LIN {X 0,Y 509.293,Z 778.89,A -85,B 0,C 180,E1 -5495.543,E2 -5495.543} C_VEL
LIN {X 0,Y 509.338,Z 774.921,A -85,B 0,C 180,E1 -5496.696,E2 -5496.696} C_VEL
LIN {X 0,Y 509.453,Z 769.669,A -85,B 0,C 180,E1 -5497.929,E2 -5497.929} C_VEL
LIN {X 0,Y 509.604,Z 763.492,A -85,B 0,C 180,E1 -5499.125,E2 -5499.125} C_VEL
LIN {X 0,Y 509.79,Z 757.418,A -85,B 0,C 180,E1 -5500.123,E2 -5500.123} C_VEL
LIN {X 0,Y 510.074,Z 750.342,A -85,B 0,C 180,E1 -5501.122,E2 -5501.122} C_VEL
LIN {X 0,Y 510.293,Z 742.434,A -85,B 0,C 180,E1 -5502.082,E2 -5502.082} C_VEL
LIN {X 0,Y 510.609,Z 734.391,A -85,B 0,C 180,E1 -5502.924,E2 -5502.924} C_VEL
LIN {X 0,Y 510.98,Z 725.51,A -85,B 0,C 180,E1 -5503.724,E2 -5503.724} C_VEL
LIN {X 0,Y 511.277,Z 716.451,A -85,B 0,C 180,E1 -5504.427,E2 -5504.427} C_VEL
LIN {X 0,Y 511.699,Z 705.64,A -85,B 0,C 180,E1 -5505.127,E2 -5505.127} C_VEL
LIN {X 0,Y 512.044,Z 695.376,A -85,B 0,C 180,E1 -5505.677,E2 -5505.677} C_VEL
LIN {X 0,Y 512.33,Z 684.979,A -85,B 0,C 180,E1 -5506.131,E2 -5506.131} C_VEL
LIN {X 0,Y 512.62,Z 672.99,A -85,B 0,C 180,E1 -5506.533,E2 -5506.533} C_VEL
LIN {X 0,Y 512.826,Z 661.767,A -85,B 0,C 180,E1 -5506.802,E2 -5506.802} C_VEL
LIN {X 0,Y 513.111,Z 631.655,A -85,B 0,C 180,E1 -5507.254,E2 -5507.254} C_VEL
LIN {X 0,Y 513.563,Z 539.81,A -85,B 0,C 180,E1 -5508.56,E2 -5508.56} C_VEL
LIN {X 0,Y 510.7,Z 525.355,A -85,B 0,C 180,E1 -5508.892,E2 -5508.892} C_VEL
LIN {X 0,Y 510.69,Z 524.406,A -85,B 0,C 180,E1 -5509.004,E2 -5509.004} C_VEL
LIN {X 0,Y 511.189,Z 507.71,A -85,B 0,C 180,E1 -5512.002,E2 -5512.002} C_VEL
LIN {X 0,Y 511.684,Z 492.965,A -85,B 0,C 180,E1 -5514.662,E2 -5514.662} C_VEL
LIN {X 0,Y 511.823,Z 486.597,A -85,B 0,C 180,E1 -5515.846,E2 -5515.846} C_VEL
LIN {X 0,Y 509.91,Z 476.204,A -85,B 0,C 180,E1 -5517.944,E2 -5517.944} C_VEL
LIN {X 0,Y 509.845,Z 476.085,A -85,B 0,C 180,E1 -5520.665,E2 -5520.665} C_VEL
LIN {X 0,Y 509.859,Z 476.102,A -85,B 0,C 180,E1 -5523.46,E2 -5523.46} C_VEL
LIN {X 0,Y 509.822,Z 476.077,A -85,B 0,C 180,E1 -5526.352,E2 -5526.352} C_VEL
LIN {X 0,Y 509.845,Z 476.1,A -85,B 0,C 180,E1 -5529.351,E2 -5529.351} C_VEL
LIN {X 0,Y 509.845,Z 476.094,A -85,B 0,C 180,E1 -5532.487,E2 -5532.487} C_VEL
LIN {X 0,Y 509.853,Z 476.102,A -85,B 0,C 180,E1 -5535.331,E2 -5535.331} C_VEL
LIN {X 0,Y 509.859,Z 476.093,A -85,B 0,C 180,E1 -5538.575,E2 -5538.575} C_VEL
LIN {X 0,Y 509.846,Z 476.096,A -85,B 0,C 180,E1 -5541.786,E2 -5541.786} C_VEL
LIN {X 0,Y 509.841,Z 476.098,A -85,B 0,C 180,E1 -5544.622,E2 -5544.622} C_VEL
LIN {X 0,Y 509.859,Z 476.098,A -85,B 0,C 180,E1 -5547.48,E2 -5547.48} C_VEL
LIN {X 0,Y 509.852,Z 476.096,A -85,B 0,C 180,E1 -5550.273,E2 -5550.273} C_VEL
LIN {X 0,Y 509.88,Z 476.09,A -85,B 0,C 180,E1 -5552.944,E2 -5552.944} C_VEL
LIN {X 0,Y 509.863,Z 476.1,A -85,B 0,C 180,E1 -5555.573,E2 -5555.573} C_VEL
LIN {X 0,Y 509.814,Z 476.096,A -85,B 0,C 180,E1 -5558.148,E2 -5558.148} C_VEL
LIN {X 0,Y 509.857,Z 476.091,A -85,B 0,C 180,E1 -5560.681,E2 -5560.681} C_VEL
LIN {X 0,Y 509.879,Z 476.098,A -85,B 0,C 180,E1 -5563.174,E2 -5563.174} C_VEL
LIN {X 0,Y 509.854,Z 476.092,A -85,B 0,C 180,E1 -5565.634,E2 -5565.634} C_VEL
LIN {X 0,Y 509.904,Z 476.089,A -85,B 0,C 180,E1 -5568.874,E2 -5568.874} C_VEL
LIN {X 0,Y 509.943,Z 476.083,A -85,B 0,C 180,E1 -5572.078,E2 -5572.078} C_VEL
LIN {X 0,Y 509.974,Z 476.07,A -85,B 0,C 180,E1 -5574.464,E2 -5574.464} C_VEL
LIN {X 0,Y 510.046,Z 476.078,A -85,B 0,C 180,E1 -5577.631,E2 -5577.631} C_VEL
LIN {X 0,Y 510.056,Z 476.066,A -85,B 0,C 180,E1 -5580.789,E2 -5580.789} C_VEL
LIN {X 0,Y 509.95,Z 476.078,A -85,B 0,C 180,E1 -5583.16,E2 -5583.16} C_VEL
LIN {X 0,Y 509.968,Z 476.081,A -85,B 0,C 180,E1 -5586.329,E2 -5586.329} C_VEL
LIN {X 0,Y 509.909,Z 476.084,A -85,B 0,C 180,E1 -5588.72,E2 -5588.72} C_VEL
LIN {X 0,Y 509.895,Z 476.093,A -85,B 0,C 180,E1 -5591.931,E2 -5591.931} C_VEL
LIN {X 0,Y 509.883,Z 476.096,A -85,B 0,C 180,E1 -5595.242,E2 -5595.242} C_VEL
LIN {X 0,Y 509.878,Z 476.092,A -85,B 0,C 180,E1 -5598.001,E2 -5598.001} C_VEL
LIN {X 0,Y 509.841,Z 476.098,A -85,B 0,C 180,E1 -5601.002,E2 -5601.002} C_VEL
LIN {X 0,Y 509.86,Z 476.088,A -85,B 0,C 180,E1 -5604.426,E2 -5604.426} C_VEL
LIN {X 0,Y 509.878,Z 476.094,A -85,B 0,C 180,E1 -5607.056,E2 -5607.056} C_VEL
LIN {X 0,Y 509.871,Z 476.094,A -85,B 0,C 180,E1 -5609.75,E2 -5609.75} C_VEL
LIN {X 0,Y 509.868,Z 476.094,A -85,B 0,C 180,E1 -5612.775,E2 -5612.775} C_VEL
LIN {X 0,Y 509.834,Z 476.102,A -85,B 0,C 180,E1 -5615.582,E2 -5615.582} C_VEL
LIN {X 0,Y 509.842,Z 476.099,A -85,B 0,C 180,E1 -5618.338,E2 -5618.338} C_VEL
LIN {X 0,Y 509.85,Z 476.096,A -85,B 0,C 180,E1 -5621.425,E2 -5621.425} C_VEL
LIN {X 0,Y 509.848,Z 476.094,A -85,B 0,C 180,E1 -5624.668,E2 -5624.668} C_VEL
LIN {X 0,Y 509.879,Z 476.092,A -85,B 0,C 180,E1 -5628.1,E2 -5628.1} C_VEL
LIN {X 0,Y 509.87,Z 476.094,A -85,B 0,C 180,E1 -5630.651,E2 -5630.651} C_VEL
LIN {X 0,Y 509.824,Z 476.095,A -85,B 0,C 180,E1 -5633.749,E2 -5633.749} C_VEL
LIN {X 0,Y 509.159,Z 476.183,A -85,B 0,C 180,E1 -5634.409,E2 -5634.409} C_VEL
LIN {X 0,Y 506.34,Z 476.537,A -85,B 0,C 180,E1 -5635.481,E2 -5635.481} C_VEL
LIN {X 0,Y 503.947,Z 476.835,A -85,B 0,C 180,E1 -5636.344,E2 -5636.344} C_VEL
LIN {X 0,Y 502.899,Z 476.964,A -85,B 0,C 180,E1 -5637.011,E2 -5637.011} C_VEL
LIN {X 0,Y 502.802,Z 476.976,A -85,B 0,C 180,E1 -5637.236,E2 -5637.236} C_VEL
LIN {X 0,Y 502.825,Z 476.978,A -85,B 0,C 180,E1 -5640.062,E2 -5640.062} C_VEL
LIN {X 0,Y 502.829,Z 476.973,A -85,B 0,C 180,E1 -5642.534,E2 -5642.534} C_VEL
LIN {X 0,Y 502.823,Z 476.975,A -85,B 0,C 180,E1 -5645.299,E2 -5645.299} C_VEL
LIN {X 0,Y 502.78,Z 476.985,A -85,B 0,C 180,E1 -5647.827,E2 -5647.827} C_VEL
LIN {X 0,Y 502.821,Z 476.976,A -85,B 0,C 180,E1 -5650.401,E2 -5650.401} C_VEL
LIN {X 0,Y 502.83,Z 476.973,A -85,B 0,C 180,E1 -5652.932,E2 -5652.932} C_VEL
LIN {X 0,Y 502.841,Z 476.974,A -85,B 0,C 180,E1 -5655.429,E2 -5655.429} C_VEL
LIN {X 0,Y 502.873,Z 476.968,A -85,B 0,C 180,E1 -5658.717,E2 -5658.717} C_VEL
LIN {X 0,Y 502.898,Z 476.97,A -85,B 0,C 180,E1 -5661.967,E2 -5661.967} C_VEL
LIN {X 0,Y 502.933,Z 476.963,A -85,B 0,C 180,E1 -5664.387,E2 -5664.387} C_VEL
LIN {X 0,Y 503.022,Z 476.953,A -85,B 0,C 180,E1 -5667.598,E2 -5667.598} C_VEL
LIN {X 0,Y 503.024,Z 476.955,A -85,B 0,C 180,E1 -5670,E2 -5670} C_VEL
LIN {X 0,Y 503.022,Z 476.953,A -85,B 0,C 180,E1 -5672.402,E2 -5672.402} C_VEL
LIN {X 0,Y 502.934,Z 476.963,A -85,B 0,C 180,E1 -5675.613,E2 -5675.613} C_VEL
LIN {X 0,Y 502.898,Z 476.97,A -85,B 0,C 180,E1 -5678.033,E2 -5678.033} C_VEL
LIN {X 0,Y 502.873,Z 476.968,A -85,B 0,C 180,E1 -5681.283,E2 -5681.283} C_VEL
LIN {X 0,Y 502.841,Z 476.974,A -85,B 0,C 180,E1 -5684.571,E2 -5684.571} C_VEL
LIN {X 0,Y 502.858,Z 476.975,A -85,B 0,C 180,E1 -5687.907,E2 -5687.907} C_VEL
LIN {X 0,Y 502.824,Z 476.976,A -85,B 0,C 180,E1 -5690.536,E2 -5690.536} C_VEL
LIN {X 0,Y 502.792,Z 476.977,A -85,B 0,C 180,E1 -5693.04,E2 -5693.04} C_VEL
LIN {X 0,Y 502.835,Z 476.975,A -85,B 0,C 180,E1 -5695.675,E2 -5695.675} C_VEL
LIN {X 0,Y 502.837,Z 476.977,A -85,B 0,C 180,E1 -5698.372,E2 -5698.372} C_VEL
LIN {X 0,Y 502.791,Z 476.978,A -85,B 0,C 180,E1 -5701.499,E2 -5701.499} C_VEL
LIN {X 0,Y 502.799,Z 476.979,A -85,B 0,C 180,E1 -5704.444,E2 -5704.444} C_VEL
LIN {X 0,Y 502.774,Z 476.969,A -85,B 0,C 180,E1 -5707.178,E2 -5707.178} C_VEL
LIN {X 0,Y 502.819,Z 476.979,A -85,B 0,C 180,E1 -5710.011,E2 -5710.011} C_VEL
LIN {X 0,Y 502.822,Z 476.963,A -85,B 0,C 180,E1 -5712.202,E2 -5712.202} C_VEL
LIN {X 0,Y 502.792,Z 476.973,A -85,B 0,C 180,E1 -5715.468,E2 -5715.468} C_VEL
LIN {X 0,Y 502.821,Z 476.976,A -85,B 0,C 180,E1 -5717.864,E2 -5717.864} C_VEL
LIN {X 0,Y 502.794,Z 476.976,A -85,B 0,C 180,E1 -5721.024,E2 -5721.024} C_VEL
LIN {X 0,Y 502.777,Z 476.979,A -85,B 0,C 180,E1 -5724.167,E2 -5724.167} C_VEL
LIN {X 0,Y 502.824,Z 476.972,A -85,B 0,C 180,E1 -5726.993,E2 -5726.993} C_VEL
LIN {X 0,Y 502.821,Z 476.97,A -85,B 0,C 180,E1 -5730.062,E2 -5730.062} C_VEL
LIN {X 0,Y 502.826,Z 476.977,A -85,B 0,C 180,E1 -5732.533,E2 -5732.533} C_VEL
LIN {X 0,Y 502.819,Z 476.965,A -85,B 0,C 180,E1 -5735.298,E2 -5735.298} C_VEL
LIN {X 0,Y 502.771,Z 476.978,A -85,B 0,C 180,E1 -5737.827,E2 -5737.827} C_VEL
LIN {X 0,Y 502.816,Z 476.977,A -85,B 0,C 180,E1 -5740.4,E2 -5740.4} C_VEL
LIN {X 0,Y 502.826,Z 476.967,A -85,B 0,C 180,E1 -5742.932,E2 -5742.932} C_VEL
LIN {X 0,Y 502.835,Z 476.969,A -85,B 0,C 180,E1 -5745.429,E2 -5745.429} C_VEL
LIN {X 0,Y 502.871,Z 476.962,A -85,B 0,C 180,E1 -5748.717,E2 -5748.717} C_VEL
LIN {X 0,Y 502.892,Z 476.96,A -85,B 0,C 180,E1 -5751.967,E2 -5751.967} C_VEL
LIN {X 0,Y 502.949,Z 476.963,A -85,B 0,C 180,E1 -5754.387,E2 -5754.387} C_VEL
LIN {X 0,Y 503.016,Z 476.937,A -85,B 0,C 180,E1 -5757.598,E2 -5757.598} C_VEL
LIN {X 0,Y 503.017,Z 476.945,A -85,B 0,C 180,E1 -5760,E2 -5760} C_VEL
LIN {X 0,Y 503.016,Z 476.954,A -85,B 0,C 180,E1 -5762.403,E2 -5762.403} C_VEL
LIN {X 0,Y 502.93,Z 476.947,A -85,B 0,C 180,E1 -5765.614,E2 -5765.614} C_VEL
LIN {X 0,Y 502.893,Z 476.962,A -85,B 0,C 180,E1 -5768.034,E2 -5768.034} C_VEL
LIN {X 0,Y 502.868,Z 476.964,A -85,B 0,C 180,E1 -5771.284,E2 -5771.284} C_VEL
LIN {X 0,Y 502.836,Z 476.969,A -85,B 0,C 180,E1 -5774.571,E2 -5774.571} C_VEL
LIN {X 0,Y 502.854,Z 476.968,A -85,B 0,C 180,E1 -5777.908,E2 -5777.908} C_VEL
LIN {X 0,Y 502.82,Z 476.971,A -85,B 0,C 180,E1 -5780.537,E2 -5780.537} C_VEL
LIN {X 0,Y 502.789,Z 476.979,A -85,B 0,C 180,E1 -5783.041,E2 -5783.041} C_VEL
LIN {X 0,Y 502.834,Z 476.968,A -85,B 0,C 180,E1 -5785.676,E2 -5785.676} C_VEL
LIN {X 0,Y 502.834,Z 476.969,A -85,B 0,C 180,E1 -5788.373,E2 -5788.373} C_VEL
LIN {X 0,Y 502.79,Z 476.974,A -85,B 0,C 180,E1 -5791.5,E2 -5791.5} C_VEL
LIN {X 0,Y 502.801,Z 476.976,A -85,B 0,C 180,E1 -5794.445,E2 -5794.445} C_VEL
LIN {X 0,Y 502.775,Z 476.976,A -85,B 0,C 180,E1 -5797.179,E2 -5797.179} C_VEL
LIN {X 0,Y 502.812,Z 476.975,A -85,B 0,C 180,E1 -5800.013,E2 -5800.013} C_VEL
LIN {X 0,Y 502.768,Z 476.982,A -85,B 0,C 180,E1 -5803.232,E2 -5803.232} C_VEL
LIN {X 0,Y 502.786,Z 476.972,A -85,B 0,C 180,E1 -5805.662,E2 -5805.662} C_VEL
LIN {X 0,Y 502.827,Z 476.968,A -85,B 0,C 180,E1 -5807.865,E2 -5807.865} C_VEL
LIN {X 0,Y 502.8,Z 476.97,A -85,B 0,C 180,E1 -5811.025,E2 -5811.025} C_VEL
LIN {X 0,Y 502.773,Z 476.957,A -85,B 0,C 180,E1 -5814.17,E2 -5814.17} C_VEL
LIN {X 0,Y 502.831,Z 476.975,A -85,B 0,C 180,E1 -5816.994,E2 -5816.994} C_VEL
LIN {X 0,Y 502.814,Z 476.967,A -85,B 0,C 180,E1 -5820.066,E2 -5820.066} C_VEL
LIN {X 0,Y 502.895,Z 477.177,A -85,B 0,C 180,E1 -5821.869,E2 -5821.869} C_VEL
LIN {X 0,Y 504.869,Z 487.556,A -85,B 0,C 180,E1 -5823.993,E2 -5823.993} C_VEL
LIN {X 0,Y 504.577,Z 499.305,A -85,B 0,C 180,E1 -5826.177,E2 -5826.177} C_VEL
LIN {X 0,Y 503.993,Z 515.407,A -85,B 0,C 180,E1 -5829.114,E2 -5829.114} C_VEL
LIN {X 0,Y 503.721,Z 524.885,A -85,B 0,C 180,E1 -5830.818,E2 -5830.818} C_VEL
LIN {X 0,Y 505.951,Z 536.372,A -85,B 0,C 180,E1 -5831.104,E2 -5831.104} C_VEL
LIN {X 0,Y 506.919,Z 541.445,A -85,B 0,C 180,E1 -5831.215,E2 -5831.215} C_VEL
LIN {X 0,Y 506.066,Z 660.21,A -85,B 0,C 180,E1 -5832.94,E2 -5832.94} C_VEL
LIN {X 0,Y 505.875,Z 671.199,A -85,B 0,C 180,E1 -5833.195,E2 -5833.195} C_VEL
LIN {X 0,Y 505.576,Z 681.524,A -85,B 0,C 180,E1 -5833.523,E2 -5833.523} C_VEL
LIN {X 0,Y 505.316,Z 691.956,A -85,B 0,C 180,E1 -5833.953,E2 -5833.953} C_VEL
LIN {X 0,Y 504.987,Z 701.932,A -85,B 0,C 180,E1 -5834.461,E2 -5834.461} C_VEL
LIN {X 0,Y 504.608,Z 711.858,A -85,B 0,C 180,E1 -5835.069,E2 -5835.069} C_VEL
LIN {X 0,Y 504.157,Z 721.586,A -85,B 0,C 180,E1 -5835.777,E2 -5835.777} C_VEL
LIN {X 0,Y 503.786,Z 731.012,A -85,B 0,C 180,E1 -5836.59,E2 -5836.59} C_VEL
LIN {X 0,Y 503.413,Z 740.042,A -85,B 0,C 180,E1 -5837.504,E2 -5837.504} C_VEL
LIN {X 0,Y 503.156,Z 747.04,A -85,B 0,C 180,E1 -5838.318,E2 -5838.318} C_VEL
LIN {X 0,Y 502.863,Z 754.543,A -85,B 0,C 180,E1 -5839.329,E2 -5839.329} C_VEL
LIN {X 0,Y 502.631,Z 761.018,A -85,B 0,C 180,E1 -5840.341,E2 -5840.341} C_VEL
LIN {X 0,Y 502.433,Z 767.557,A -85,B 0,C 180,E1 -5841.554,E2 -5841.554} C_VEL
LIN {X 0,Y 502.254,Z 772.985,A -85,B 0,C 180,E1 -5842.765,E2 -5842.765} C_VEL
LIN {X 0,Y 502.193,Z 777.426,A -85,B 0,C 180,E1 -5843.975,E2 -5843.975} C_VEL
LIN {X 0,Y 502.103,Z 780.963,A -85,B 0,C 180,E1 -5845.183,E2 -5845.183} C_VEL
LIN {X 0,Y 502.112,Z 782.9,A -85,B 0,C 180,E1 -5845.987,E2 -5845.987} C_VEL
LIN {X 0,Y 502.089,Z 785.576,A -85,B 0,C 180,E1 -5847.593,E2 -5847.593} C_VEL
LIN {X 0,Y 501.988,Z 786.858,A -85,B 0,C 180,E1 -5849.198,E2 -5849.198} C_VEL
LIN {X 0,Y 501.979,Z 787.109,A -85,B 0,C 180,E1 -5850,E2 -5850} C_VEL
LIN {X 0,Y 502.033,Z 786.388,A -85,B 0,C 180,E1 -5851.604,E2 -5851.604} C_VEL
LIN {X 0,Y 502.089,Z 785.576,A -85,B 0,C 180,E1 -5852.407,E2 -5852.407} C_VEL
LIN {X 0,Y 502.112,Z 782.9,A -85,B 0,C 180,E1 -5854.013,E2 -5854.013} C_VEL
LIN {X 0,Y 502.205,Z 778.691,A -85,B 0,C 180,E1 -5855.622,E2 -5855.622} C_VEL
LIN {X 0,Y 502.259,Z 774.722,A -85,B 0,C 180,E1 -5856.79,E2 -5856.79} C_VEL
LIN {X 0,Y 502.382,Z 769.469,A -85,B 0,C 180,E1 -5858.041,E2 -5858.041} C_VEL
LIN {X 0,Y 502.562,Z 763.293,A -85,B 0,C 180,E1 -5859.254,E2 -5859.254} C_VEL
LIN {X 0,Y 502.736,Z 757.218,A -85,B 0,C 180,E1 -5860.267,E2 -5860.267} C_VEL
LIN {X 0,Y 503.042,Z 750.142,A -85,B 0,C 180,E1 -5861.279,E2 -5861.279} C_VEL
LIN {X 0,Y 503.31,Z 742.041,A -85,B 0,C 180,E1 -5862.274,E2 -5862.274} C_VEL
LIN {X 0,Y 503.684,Z 733.132,A -85,B 0,C 180,E1 -5863.207,E2 -5863.207} C_VEL
LIN {X 0,Y 504.049,Z 724.068,A -85,B 0,C 180,E1 -5864.02,E2 -5864.02} C_VEL
LIN {X 0,Y 504.425,Z 714.786,A -85,B 0,C 180,E1 -5864.73,E2 -5864.73} C_VEL
LIN {X 0,Y 504.826,Z 705.441,A -85,B 0,C 180,E1 -5865.338,E2 -5865.338} C_VEL
LIN {X 0,Y 505.189,Z 695.177,A -85,B 0,C 180,E1 -5865.895,E2 -5865.895} C_VEL
LIN {X 0,Y 505.521,Z 684.654,A -85,B 0,C 180,E1 -5866.359,E2 -5866.359} C_VEL
LIN {X 0,Y 505.796,Z 673.229,A -85,B 0,C 180,E1 -5866.75,E2 -5866.75} C_VEL
LIN {X 0,Y 506.053,Z 661.57,A -85,B 0,C 180,E1 -5867.034,E2 -5867.034} C_VEL
LIN {X 0,Y 506.35,Z 631.458,A -85,B 0,C 180,E1 -5867.492,E2 -5867.492} C_VEL
LIN {X 0,Y 506.814,Z 540.888,A -85,B 0,C 180,E1 -5868.797,E2 -5868.797} C_VEL
LIN {X 0,Y 503.72,Z 525.076,A -85,B 0,C 180,E1 -5869.168,E2 -5869.168} C_VEL
LIN {X 0,Y 503.786,Z 522.695,A -85,B 0,C 180,E1 -5869.56,E2 -5869.56} C_VEL
LIN {X 0,Y 504.263,Z 507.55,A -85,B 0,C 180,E1 -5872.32,E2 -5872.32} C_VEL
LIN {X 0,Y 504.863,Z 491.859,A -85,B 0,C 180,E1 -5875.198,E2 -5875.198} C_VEL
LIN {X 0,Y 504.725,Z 486.455,A -85,B 0,C 180,E1 -5876.237,E2 -5876.237} C_VEL
LIN {X 0,Y 502.93,Z 477.303,A -85,B 0,C 180,E1 -5878.101,E2 -5878.101} C_VEL
LIN {X 0,Y 502.84,Z 476.965,A -85,B 0,C 180,E1 -5878.372,E2 -5878.372} C_VEL
LIN {X 0,Y 502.794,Z 476.965,A -85,B 0,C 180,E1 -5881.499,E2 -5881.499} C_VEL
LIN {X 0,Y 502.803,Z 476.976,A -85,B 0,C 180,E1 -5883.993,E2 -5883.993} C_VEL
LIN {X 0,Y 502.775,Z 476.956,A -85,B 0,C 180,E1 -5887.177,E2 -5887.177} C_VEL
LIN {X 0,Y 502.786,Z 476.977,A -85,B 0,C 180,E1 -5890.014,E2 -5890.014} C_VEL
LIN {X 0,Y 502.8,Z 476.971,A -85,B 0,C 180,E1 -5892.198,E2 -5892.198} C_VEL
LIN {X 0,Y 502.797,Z 476.981,A -85,B 0,C 180,E1 -5895.467,E2 -5895.467} C_VEL
LIN {X 0,Y 502.822,Z 476.973,A -85,B 0,C 180,E1 -5898.934,E2 -5898.934} C_VEL
LIN {X 0,Y 502.789,Z 476.973,A -85,B 0,C 180,E1 -5902.045,E2 -5902.045} C_VEL
LIN {X 0,Y 502.804,Z 476.979,A -85,B 0,C 180,E1 -5905.034,E2 -5905.034} C_VEL
LIN {X 0,Y 502.781,Z 476.977,A -85,B 0,C 180,E1 -5907.915,E2 -5907.915} C_VEL
LIN {X 0,Y 502.818,Z 476.973,A -85,B 0,C 180,E1 -5910.711,E2 -5910.711} C_VEL
LIN {X 0,Y 502.874,Z 476.966,A -85,B 0,C 180,E1 -5913.434,E2 -5913.434} C_VEL
LIN {X 0,Y 502.784,Z 476.977,A -85,B 0,C 180,E1 -5916.086,E2 -5916.086} C_VEL
LIN {X 0,Y 502.776,Z 476.973,A -85,B 0,C 180,E1 -5918.688,E2 -5918.688} C_VEL
LIN {X 0,Y 502.823,Z 476.973,A -85,B 0,C 180,E1 -5921.248,E2 -5921.248} C_VEL
LIN {X 0,Y 502.815,Z 476.974,A -85,B 0,C 180,E1 -5923.767,E2 -5923.767} C_VEL
LIN {X 0,Y 502.822,Z 476.961,A -85,B 0,C 180,E1 -5926.254,E2 -5926.254} C_VEL
LIN {X 0,Y 502.868,Z 476.964,A -85,B 0,C 180,E1 -5928.716,E2 -5928.716} C_VEL
LIN {X 0,Y 502.893,Z 476.962,A -85,B 0,C 180,E1 -5931.966,E2 -5931.966} C_VEL
LIN {X 0,Y 502.93,Z 476.947,A -85,B 0,C 180,E1 -5934.386,E2 -5934.386} C_VEL
LIN {X 0,Y 503.016,Z 476.954,A -85,B 0,C 180,E1 -5937.597,E2 -5937.597} C_VEL
LIN {X 0,Y 503.017,Z 476.945,A -85,B 0,C 180,E1 -5940,E2 -5940} C_VEL
LIN {X 0,Y 503.016,Z 476.937,A -85,B 0,C 180,E1 -5942.402,E2 -5942.402} C_VEL
LIN {X 0,Y 502.929,Z 476.965,A -85,B 0,C 180,E1 -5945.613,E2 -5945.613} C_VEL
LIN {X 0,Y 502.892,Z 476.96,A -85,B 0,C 180,E1 -5948.033,E2 -5948.033} C_VEL
LIN {X 0,Y 502.871,Z 476.962,A -85,B 0,C 180,E1 -5951.283,E2 -5951.283} C_VEL
LIN {X 0,Y 502.835,Z 476.969,A -85,B 0,C 180,E1 -5954.571,E2 -5954.571} C_VEL
LIN {X 0,Y 502.852,Z 476.968,A -85,B 0,C 180,E1 -5957.907,E2 -5957.907} C_VEL
LIN {X 0,Y 502.818,Z 476.972,A -85,B 0,C 180,E1 -5960.536,E2 -5960.536} C_VEL
LIN {X 0,Y 502.784,Z 476.975,A -85,B 0,C 180,E1 -5963.04,E2 -5963.04} C_VEL
LIN {X 0,Y 502.832,Z 476.973,A -85,B 0,C 180,E1 -5965.676,E2 -5965.676} C_VEL
LIN {X 0,Y 502.833,Z 476.97,A -85,B 0,C 180,E1 -5968.373,E2 -5968.373} C_VEL
LIN {X 0,Y 502.788,Z 476.975,A -85,B 0,C 180,E1 -5971.5,E2 -5971.5} C_VEL
LIN {X 0,Y 502.798,Z 476.974,A -85,B 0,C 180,E1 -5974.445,E2 -5974.445} C_VEL
LIN {X 0,Y 502.772,Z 476.977,A -85,B 0,C 180,E1 -5977.179,E2 -5977.179} C_VEL
LIN {X 0,Y 502.779,Z 476.977,A -85,B 0,C 180,E1 -5980.015,E2 -5980.015} C_VEL
LIN {X 0,Y 502.821,Z 476.975,A -85,B 0,C 180,E1 -5982.203,E2 -5982.203} C_VEL
LIN {X 0,Y 502.793,Z 476.975,A -85,B 0,C 180,E1 -5985.468,E2 -5985.468} C_VEL
LIN {X 0,Y 502.831,Z 476.964,A -85,B 0,C 180,E1 -5987.866,E2 -5987.866} C_VEL
LIN {X 0,Y 502.814,Z 476.974,A -85,B 0,C 180,E1 -5991.026,E2 -5991.026} C_VEL
LIN {X 0,Y 502.779,Z 476.978,A -85,B 0,C 180,E1 -5994.168,E2 -5994.168} C_VEL
LIN {X 0,Y 502.802,Z 476.976,A -85,B 0,C 180,E1 -5997.236,E2 -5997.236} C_VEL
LIN {X 0,Y 502.105,Z 477.069,A -85,B 0,C 180,E1 -5997.905,E2 -5997.905} C_VEL
LIN {X 0,Y 499.247,Z 477.421,A -85,B 0,C 180,E1 -5998.991,E2 -5998.991} C_VEL
LIN {X 0,Y 496.855,Z 477.723,A -85,B 0,C 180,E1 -5999.866,E2 -5999.866} C_VEL
LIN {X 0,Y 495.838,Z 477.844,A -85,B 0,C 180,E1 -6000.542,E2 -6000.542} C_VEL
LIN {X 0,Y 495.759,Z 477.853,A -85,B 0,C 180,E1 -6000.77,E2 -6000.77} C_VEL
LIN {X 0,Y 495.786,Z 477.856,A -85,B 0,C 180,E1 -6003.933,E2 -6003.933} C_VEL
LIN {X 0,Y 495.76,Z 477.854,A -85,B 0,C 180,E1 -6007.138,E2 -6007.138} C_VEL
LIN {X 0,Y 495.768,Z 477.858,A -85,B 0,C 180,E1 -6010.11,E2 -6010.11} C_VEL
LIN {X 0,Y 495.782,Z 477.852,A -85,B 0,C 180,E1 -6012.682,E2 -6012.682} C_VEL
LIN {X 0,Y 495.786,Z 477.852,A -85,B 0,C 180,E1 -6015.217,E2 -6015.217} C_VEL
LIN {X 0,Y 495.848,Z 477.844,A -85,B 0,C 180,E1 -6018.555,E2 -6018.555} C_VEL
LIN {X 0,Y 495.869,Z 477.845,A -85,B 0,C 180,E1 -6021.852,E2 -6021.852} C_VEL
LIN {X 0,Y 495.891,Z 477.841,A -85,B 0,C 180,E1 -6024.307,E2 -6024.307} C_VEL
LIN {X 0,Y 495.991,Z 477.829,A -85,B 0,C 180,E1 -6027.564,E2 -6027.564} C_VEL
LIN {X 0,Y 495.996,Z 477.831,A -85,B 0,C 180,E1 -6030,E2 -6030} C_VEL
LIN {X 0,Y 495.991,Z 477.829,A -85,B 0,C 180,E1 -6032.436,E2 -6032.436} C_VEL
LIN {X 0,Y 495.892,Z 477.841,A -85,B 0,C 180,E1 -6035.693,E2 -6035.693} C_VEL
LIN {X 0,Y 495.869,Z 477.846,A -85,B 0,C 180,E1 -6038.148,E2 -6038.148} C_VEL
LIN {X 0,Y 495.848,Z 477.844,A -85,B 0,C 180,E1 -6041.445,E2 -6041.445} C_VEL
LIN {X 0,Y 495.786,Z 477.852,A -85,B 0,C 180,E1 -6044.783,E2 -6044.783} C_VEL
LIN {X 0,Y 495.782,Z 477.852,A -85,B 0,C 180,E1 -6047.318,E2 -6047.318} C_VEL
LIN {X 0,Y 495.768,Z 477.858,A -85,B 0,C 180,E1 -6049.89,E2 -6049.89} C_VEL
LIN {X 0,Y 495.76,Z 477.854,A -85,B 0,C 180,E1 -6052.862,E2 -6052.862} C_VEL
LIN {X 0,Y 495.786,Z 477.856,A -85,B 0,C 180,E1 -6056.067,E2 -6056.067} C_VEL
LIN {X 0,Y 495.774,Z 477.852,A -85,B 0,C 180,E1 -6058.814,E2 -6058.814} C_VEL
LIN {X 0,Y 495.753,Z 477.857,A -85,B 0,C 180,E1 -6061.726,E2 -6061.726} C_VEL
LIN {X 0,Y 495.769,Z 477.851,A -85,B 0,C 180,E1 -6064.695,E2 -6064.695} C_VEL
LIN {X 0,Y 495.726,Z 477.848,A -85,B 0,C 180,E1 -6067.561,E2 -6067.561} C_VEL
LIN {X 0,Y 495.786,Z 477.855,A -85,B 0,C 180,E1 -6070.052,E2 -6070.052} C_VEL
LIN {X 0,Y 495.756,Z 477.834,A -85,B 0,C 180,E1 -6072.879,E2 -6072.879} C_VEL
LIN {X 0,Y 495.728,Z 477.858,A -85,B 0,C 180,E1 -6075.999,E2 -6075.999} C_VEL
LIN {X 0,Y 495.755,Z 477.85,A -85,B 0,C 180,E1 -6078.706,E2 -6078.706} C_VEL
LIN {X 0,Y 495.742,Z 477.854,A -85,B 0,C 180,E1 -6081.408,E2 -6081.408} C_VEL
LIN {X 0,Y 495.749,Z 477.855,A -85,B 0,C 180,E1 -6084.463,E2 -6084.463} C_VEL
LIN {X 0,Y 495.76,Z 477.851,A -85,B 0,C 180,E1 -6087.406,E2 -6087.406} C_VEL
LIN {X 0,Y 495.772,Z 477.849,A -85,B 0,C 180,E1 -6090.255,E2 -6090.255} C_VEL
LIN {X 0,Y 495.824,Z 477.843,A -85,B 0,C 180,E1 -6093.248,E2 -6093.248} C_VEL
LIN {X 0,Y 495.742,Z 477.847,A -85,B 0,C 180,E1 -6095.725,E2 -6095.725} C_VEL
LIN {X 0,Y 495.733,Z 477.862,A -85,B 0,C 180,E1 -6098.371,E2 -6098.371} C_VEL
LIN {X 0,Y 495.775,Z 477.846,A -85,B 0,C 180,E1 -6100.972,E2 -6100.972} C_VEL
LIN {X 0,Y 495.771,Z 477.843,A -85,B 0,C 180,E1 -6103.53,E2 -6103.53} C_VEL
LIN {X 0,Y 495.784,Z 477.852,A -85,B 0,C 180,E1 -6106.056,E2 -6106.056} C_VEL
LIN {X 0,Y 495.845,Z 477.84,A -85,B 0,C 180,E1 -6108.555,E2 -6108.555} C_VEL
LIN {X 0,Y 495.864,Z 477.834,A -85,B 0,C 180,E1 -6111.852,E2 -6111.852} C_VEL
LIN {X 0,Y 495.904,Z 477.839,A -85,B 0,C 180,E1 -6114.307,E2 -6114.307} C_VEL
LIN {X 0,Y 495.985,Z 477.812,A -85,B 0,C 180,E1 -6117.564,E2 -6117.564} C_VEL
LIN {X 0,Y 495.988,Z 477.82,A -85,B 0,C 180,E1 -6120,E2 -6120} C_VEL
LIN {X 0,Y 495.985,Z 477.83,A -85,B 0,C 180,E1 -6122.437,E2 -6122.437} C_VEL
LIN {X 0,Y 495.888,Z 477.824,A -85,B 0,C 180,E1 -6125.694,E2 -6125.694} C_VEL
LIN {X 0,Y 495.864,Z 477.838,A -85,B 0,C 180,E1 -6128.148,E2 -6128.148} C_VEL
LIN {X 0,Y 495.842,Z 477.838,A -85,B 0,C 180,E1 -6131.446,E2 -6131.446} C_VEL
LIN {X 0,Y 495.781,Z 477.851,A -85,B 0,C 180,E1 -6134.783,E2 -6134.783} C_VEL
LIN {X 0,Y 495.779,Z 477.849,A -85,B 0,C 180,E1 -6137.319,E2 -6137.319} C_VEL
LIN {X 0,Y 495.77,Z 477.846,A -85,B 0,C 180,E1 -6139.891,E2 -6139.891} C_VEL
LIN {X 0,Y 495.75,Z 477.858,A -85,B 0,C 180,E1 -6142.861,E2 -6142.861} C_VEL
LIN {X 0,Y 495.792,Z 477.847,A -85,B 0,C 180,E1 -6146.068,E2 -6146.068} C_VEL
LIN {X 0,Y 495.766,Z 477.857,A -85,B 0,C 180,E1 -6148.815,E2 -6148.815} C_VEL
LIN {X 0,Y 495.752,Z 477.851,A -85,B 0,C 180,E1 -6151.727,E2 -6151.727} C_VEL
LIN {X 0,Y 495.771,Z 477.855,A -85,B 0,C 180,E1 -6154.696,E2 -6154.696} C_VEL
LIN {X 0,Y 495.726,Z 477.852,A -85,B 0,C 180,E1 -6157.562,E2 -6157.562} C_VEL
LIN {X 0,Y 495.773,Z 477.857,A -85,B 0,C 180,E1 -6160.7,E2 -6160.7} C_VEL
LIN {X 0,Y 495.729,Z 477.857,A -85,B 0,C 180,E1 -6164.002,E2 -6164.002} C_VEL
LIN {X 0,Y 495.73,Z 477.852,A -85,B 0,C 180,E1 -6167.119,E2 -6167.119} C_VEL
LIN {X 0,Y 495.757,Z 477.853,A -85,B 0,C 180,E1 -6169.954,E2 -6169.954} C_VEL
LIN {X 0,Y 495.725,Z 477.836,A -85,B 0,C 180,E1 -6172.554,E2 -6172.554} C_VEL
LIN {X 0,Y 495.777,Z 477.852,A -85,B 0,C 180,E1 -6175.458,E2 -6175.458} C_VEL
LIN {X 0,Y 495.757,Z 477.842,A -85,B 0,C 180,E1 -6178.365,E2 -6178.365} C_VEL
LIN {X 0,Y 495.818,Z 478.011,A -85,B 0,C 180,E1 -6181.622,E2 -6181.622} C_VEL
LIN {X 0,Y 497.902,Z 488.588,A -85,B 0,C 180,E1 -6183.827,E2 -6183.827} C_VEL
LIN {X 0,Y 497.785,Z 496.786,A -85,B 0,C 180,E1 -6185.387,E2 -6185.387} C_VEL
LIN {X 0,Y 497.17,Z 513.2,A -85,B 0,C 180,E1 -6188.437,E2 -6188.437} C_VEL
LIN {X 0,Y 496.762,Z 524.802,A -85,B 0,C 180,E1 -6190.548,E2 -6190.548} C_VEL
LIN {X 0,Y 500.191,Z 542.269,A -85,B 0,C 180,E1 -6190.968,E2 -6190.968} C_VEL
LIN {X 0,Y 499.297,Z 660.012,A -85,B 0,C 180,E1 -6192.702,E2 -6192.702} C_VEL
LIN {X 0,Y 499.05,Z 670.783,A -85,B 0,C 180,E1 -6192.952,E2 -6192.952} C_VEL
LIN {X 0,Y 498.773,Z 681.506,A -85,B 0,C 180,E1 -6193.299,E2 -6193.299} C_VEL
LIN {X 0,Y 498.483,Z 691.757,A -85,B 0,C 180,E1 -6193.727,E2 -6193.727} C_VEL
LIN {X 0,Y 498.102,Z 701.733,A -85,B 0,C 180,E1 -6194.24,E2 -6194.24} C_VEL
LIN {X 0,Y 497.713,Z 711.659,A -85,B 0,C 180,E1 -6194.857,E2 -6194.857} C_VEL
LIN {X 0,Y 497.224,Z 721.386,A -85,B 0,C 180,E1 -6195.575,E2 -6195.575} C_VEL
LIN {X 0,Y 496.799,Z 730.811,A -85,B 0,C 180,E1 -6196.398,E2 -6196.398} C_VEL
LIN {X 0,Y 496.42,Z 739.838,A -85,B 0,C 180,E1 -6197.324,E2 -6197.324} C_VEL
LIN {X 0,Y 496.12,Z 747.179,A -85,B 0,C 180,E1 -6198.195,E2 -6198.195} C_VEL
LIN {X 0,Y 495.829,Z 754.343,A -85,B 0,C 180,E1 -6199.175,E2 -6199.175} C_VEL
LIN {X 0,Y 495.546,Z 761.956,A -85,B 0,C 180,E1 -6200.408,E2 -6200.408} C_VEL
LIN {X 0,Y 495.385,Z 767.358,A -85,B 0,C 180,E1 -6201.433,E2 -6201.433} C_VEL
LIN {X 0,Y 495.18,Z 772.786,A -85,B 0,C 180,E1 -6202.661,E2 -6202.661} C_VEL
LIN {X 0,Y 495.112,Z 776.862,A -85,B 0,C 180,E1 -6203.771,E2 -6203.771} C_VEL
LIN {X 0,Y 495.03,Z 780.765,A -85,B 0,C 180,E1 -6205.114,E2 -6205.114} C_VEL
LIN {X 0,Y 495.009,Z 782.701,A -85,B 0,C 180,E1 -6205.929,E2 -6205.929} C_VEL
LIN {X 0,Y 494.995,Z 785.378,A -85,B 0,C 180,E1 -6207.559,E2 -6207.559} C_VEL
LIN {X 0,Y 494.908,Z 786.661,A -85,B 0,C 180,E1 -6209.186,E2 -6209.186} C_VEL
LIN {X 0,Y 494.896,Z 786.912,A -85,B 0,C 180,E1 -6210,E2 -6210} C_VEL
LIN {X 0,Y 494.959,Z 786.191,A -85,B 0,C 180,E1 -6211.627,E2 -6211.627} C_VEL
LIN {X 0,Y 494.995,Z 785.378,A -85,B 0,C 180,E1 -6212.441,E2 -6212.441} C_VEL
LIN {X 0,Y 495.009,Z 782.701,A -85,B 0,C 180,E1 -6214.071,E2 -6214.071} C_VEL
LIN {X 0,Y 495.102,Z 779.753,A -85,B 0,C 180,E1 -6215.294,E2 -6215.294} C_VEL
LIN {X 0,Y 495.129,Z 775.931,A -85,B 0,C 180,E1 -6216.52,E2 -6216.52} C_VEL
LIN {X 0,Y 495.24,Z 771.173,A -85,B 0,C 180,E1 -6217.748,E2 -6217.748} C_VEL
LIN {X 0,Y 495.451,Z 764.231,A -85,B 0,C 180,E1 -6219.182,E2 -6219.182} C_VEL
LIN {X 0,Y 495.713,Z 757.019,A -85,B 0,C 180,E1 -6220.414,E2 -6220.414} C_VEL
LIN {X 0,Y 496.012,Z 749.942,A -85,B 0,C 180,E1 -6221.441,E2 -6221.441} C_VEL
LIN {X 0,Y 496.259,Z 743.477,A -85,B 0,C 180,E1 -6222.264,E2 -6222.264} C_VEL
LIN {X 0,Y 496.671,Z 733.992,A -85,B 0,C 180,E1 -6223.293,E2 -6223.293} C_VEL
LIN {X 0,Y 497.079,Z 725.11,A -85,B 0,C 180,E1 -6224.116,E2 -6224.116} C_VEL
LIN {X 0,Y 497.484,Z 716.053,A -85,B 0,C 180,E1 -6224.836,E2 -6224.836} C_VEL
LIN {X 0,Y 497.963,Z 705.242,A -85,B 0,C 180,E1 -6225.554,E2 -6225.554} C_VEL
LIN {X 0,Y 498.348,Z 694.979,A -85,B 0,C 180,E1 -6226.119,E2 -6226.119} C_VEL
LIN {X 0,Y 498.696,Z 684.122,A -85,B 0,C 180,E1 -6226.603,E2 -6226.603} C_VEL
LIN {X 0,Y 499.053,Z 672.572,A -85,B 0,C 180,E1 -6226.997,E2 -6226.997} C_VEL
LIN {X 0,Y 499.289,Z 661.372,A -85,B 0,C 180,E1 -6227.272,E2 -6227.272} C_VEL
LIN {X 0,Y 499.566,Z 633.05,A -85,B 0,C 180,E1 -6227.711,E2 -6227.711} C_VEL
LIN {X 0,Y 500.19,Z 542.447,A -85,B 0,C 180,E1 -6229.03,E2 -6229.03} C_VEL
LIN {X 0,Y 496.726,Z 524.746,A -85,B 0,C 180,E1 -6229.457,E2 -6229.457} C_VEL
LIN {X 0,Y 497.296,Z 509.746,A -85,B 0,C 180,E1 -6232.212,E2 -6232.212} C_VEL
LIN {X 0,Y 497.86,Z 494.427,A -85,B 0,C 180,E1 -6235.055,E2 -6235.055} C_VEL
LIN {X 0,Y 497.893,Z 488.621,A -85,B 0,C 180,E1 -6236.174,E2 -6236.174} C_VEL
LIN {X 0,Y 495.808,Z 477.951,A -85,B 0,C 180,E1 -6238.415,E2 -6238.415} C_VEL
LIN {X 0,Y 495.757,Z 477.843,A -85,B 0,C 180,E1 -6241.725,E2 -6241.725} C_VEL
LIN {X 0,Y 495.768,Z 477.849,A -85,B 0,C 180,E1 -6244.693,E2 -6244.693} C_VEL
LIN {X 0,Y 495.726,Z 477.838,A -85,B 0,C 180,E1 -6247.561,E2 -6247.561} C_VEL
LIN {X 0,Y 495.764,Z 477.854,A -85,B 0,C 180,E1 -6250.699,E2 -6250.699} C_VEL
LIN {X 0,Y 495.731,Z 477.852,A -85,B 0,C 180,E1 -6253.695,E2 -6253.695} C_VEL
LIN {X 0,Y 495.724,Z 477.857,A -85,B 0,C 180,E1 -6256.305,E2 -6256.305} C_VEL
LIN {X 0,Y 495.773,Z 477.857,A -85,B 0,C 180,E1 -6259.3,E2 -6259.3} C_VEL
LIN {X 0,Y 495.726,Z 477.852,A -85,B 0,C 180,E1 -6262.438,E2 -6262.438} C_VEL
LIN {X 0,Y 495.779,Z 477.852,A -85,B 0,C 180,E1 -6265.457,E2 -6265.457} C_VEL
LIN {X 0,Y 495.752,Z 477.851,A -85,B 0,C 180,E1 -6268.363,E2 -6268.363} C_VEL
LIN {X 0,Y 495.781,Z 477.849,A -85,B 0,C 180,E1 -6271.506,E2 -6271.506} C_VEL
LIN {X 0,Y 495.792,Z 477.847,A -85,B 0,C 180,E1 -6273.932,E2 -6273.932} C_VEL
LIN {X 0,Y 495.75,Z 477.858,A -85,B 0,C 180,E1 -6277.139,E2 -6277.139} C_VEL
LIN {X 0,Y 495.77,Z 477.846,A -85,B 0,C 180,E1 -6280.109,E2 -6280.109} C_VEL
LIN {X 0,Y 495.78,Z 477.849,A -85,B 0,C 180,E1 -6282.681,E2 -6282.681} C_VEL
LIN {X 0,Y 495.781,Z 477.851,A -85,B 0,C 180,E1 -6285.217,E2 -6285.217} C_VEL
LIN {X 0,Y 495.842,Z 477.838,A -85,B 0,C 180,E1 -6288.554,E2 -6288.554} C_VEL
LIN {X 0,Y 495.864,Z 477.838,A -85,B 0,C 180,E1 -6291.852,E2 -6291.852} C_VEL
LIN {X 0,Y 495.888,Z 477.824,A -85,B 0,C 180,E1 -6294.306,E2 -6294.306} C_VEL
LIN {X 0,Y 495.985,Z 477.83,A -85,B 0,C 180,E1 -6297.563,E2 -6297.563} C_VEL
LIN {X 0,Y 495.988,Z 477.82,A -85,B 0,C 180,E1 -6300,E2 -6300} C_VEL
LIN {X 0,Y 495.985,Z 477.812,A -85,B 0,C 180,E1 -6302.436,E2 -6302.436} C_VEL
LIN {X 0,Y 495.887,Z 477.841,A -85,B 0,C 180,E1 -6305.693,E2 -6305.693} C_VEL
LIN {X 0,Y 495.864,Z 477.834,A -85,B 0,C 180,E1 -6308.148,E2 -6308.148} C_VEL
LIN {X 0,Y 495.845,Z 477.84,A -85,B 0,C 180,E1 -6311.445,E2 -6311.445} C_VEL
LIN {X 0,Y 495.78,Z 477.849,A -85,B 0,C 180,E1 -6314.783,E2 -6314.783} C_VEL
LIN {X 0,Y 495.778,Z 477.846,A -85,B 0,C 180,E1 -6317.318,E2 -6317.318} C_VEL
LIN {X 0,Y 495.769,Z 477.855,A -85,B 0,C 180,E1 -6319.89,E2 -6319.89} C_VEL
LIN {X 0,Y 495.751,Z 477.85,A -85,B 0,C 180,E1 -6322.861,E2 -6322.861} C_VEL
LIN {X 0,Y 495.79,Z 477.85,A -85,B 0,C 180,E1 -6326.067,E2 -6326.067} C_VEL
LIN {X 0,Y 495.771,Z 477.849,A -85,B 0,C 180,E1 -6328.814,E2 -6328.814} C_VEL
LIN {X 0,Y 495.75,Z 477.856,A -85,B 0,C 180,E1 -6331.726,E2 -6331.726} C_VEL
LIN {X 0,Y 495.768,Z 477.849,A -85,B 0,C 180,E1 -6334.696,E2 -6334.696} C_VEL
LIN {X 0,Y 495.723,Z 477.86,A -85,B 0,C 180,E1 -6337.562,E2 -6337.562} C_VEL
LIN {X 0,Y 495.758,Z 477.847,A -85,B 0,C 180,E1 -6340.7,E2 -6340.7} C_VEL
LIN {X 0,Y 495.726,Z 477.863,A -85,B 0,C 180,E1 -6343.696,E2 -6343.696} C_VEL
LIN {X 0,Y 495.727,Z 477.838,A -85,B 0,C 180,E1 -6346.305,E2 -6346.305} C_VEL
LIN {X 0,Y 495.779,Z 477.849,A -85,B 0,C 180,E1 -6349.303,E2 -6349.303} C_VEL
LIN {X 0,Y 495.757,Z 477.856,A -85,B 0,C 180,E1 -6351.41,E2 -6351.41} C_VEL
LIN {X 0,Y 495.751,Z 477.853,A -85,B 0,C 180,E1 -6354.463,E2 -6354.463} C_VEL
LIN {X 0,Y 495.763,Z 477.856,A -85,B 0,C 180,E1 -6357.406,E2 -6357.406} C_VEL
LIN {X 0,Y 495.776,Z 477.854,A -85,B 0,C 180,E1 -6360.255,E2 -6360.255} C_VEL
LIN {X 0,Y 495.759,Z 477.853,A -85,B 0,C 180,E1 -6360.77,E2 -6360.77} C_VEL
LIN {X 0,Y 495.098,Z 477.94,A -85,B 0,C 180,E1 -6361.449,E2 -6361.449} C_VEL
LIN {X 0,Y 492.236,Z 478.293,A -85,B 0,C 180,E1 -6362.552,E2 -6362.552} C_VEL
LIN {X 0,Y 489.826,Z 478.596,A -85,B 0,C 180,E1 -6363.44,E2 -6363.44} C_VEL
LIN {X 0,Y 488.81,Z 478.724,A -85,B 0,C 180,E1 -6364.126,E2 -6364.126} C_VEL
LIN {X 0,Y 488.738,Z 478.729,A -85,B 0,C 180,E1 -6364.359,E2 -6364.359} C_VEL
LIN {X 0,Y 488.723,Z 478.731,A -85,B 0,C 180,E1 -6367.154,E2 -6367.154} C_VEL
LIN {X 0,Y 488.721,Z 478.736,A -85,B 0,C 180,E1 -6369.811,E2 -6369.811} C_VEL
LIN {X 0,Y 488.73,Z 478.732,A -85,B 0,C 180,E1 -6372.424,E2 -6372.424} C_VEL
LIN {X 0,Y 488.758,Z 478.727,A -85,B 0,C 180,E1 -6375,E2 -6375} C_VEL
LIN {X 0,Y 488.802,Z 478.724,A -85,B 0,C 180,E1 -6378.388,E2 -6378.388} C_VEL
LIN {X 0,Y 488.814,Z 478.724,A -85,B 0,C 180,E1 -6381.734,E2 -6381.734} C_VEL
LIN {X 0,Y 488.851,Z 478.719,A -85,B 0,C 180,E1 -6384.224,E2 -6384.224} C_VEL
LIN {X 0,Y 488.958,Z 478.705,A -85,B 0,C 180,E1 -6387.529,E2 -6387.529} C_VEL
LIN {X 0,Y 488.951,Z 478.704,A -85,B 0,C 180,E1 -6390.824,E2 -6390.824} C_VEL
LIN {X 0,Y 488.958,Z 478.705,A -85,B 0,C 180,E1 -6392.471,E2 -6392.471} C_VEL
LIN {X 0,Y 488.851,Z 478.719,A -85,B 0,C 180,E1 -6395.776,E2 -6395.776} C_VEL
LIN {X 0,Y 488.814,Z 478.724,A -85,B 0,C 180,E1 -6398.266,E2 -6398.266} C_VEL
LIN {X 0,Y 488.802,Z 478.724,A -85,B 0,C 180,E1 -6401.612,E2 -6401.612} C_VEL
LIN {X 0,Y 488.758,Z 478.727,A -85,B 0,C 180,E1 -6405,E2 -6405} C_VEL
LIN {X 0,Y 488.75,Z 478.731,A -85,B 0,C 180,E1 -6408.442,E2 -6408.442} C_VEL
LIN {X 0,Y 488.702,Z 478.733,A -85,B 0,C 180,E1 -6411.07,E2 -6411.07} C_VEL
LIN {X 0,Y 488.689,Z 478.738,A -85,B 0,C 180,E1 -6413.745,E2 -6413.745} C_VEL
LIN {X 0,Y 488.786,Z 478.723,A -85,B 0,C 180,E1 -6416.943,E2 -6416.943} C_VEL
LIN {X 0,Y 488.728,Z 478.736,A -85,B 0,C 180,E1 -6420.218,E2 -6420.218} C_VEL
LIN {X 0,Y 488.729,Z 478.73,A -85,B 0,C 180,E1 -6423.484,E2 -6423.484} C_VEL
LIN {X 0,Y 488.682,Z 478.726,A -85,B 0,C 180,E1 -6426.355,E2 -6426.355} C_VEL
LIN {X 0,Y 488.741,Z 478.727,A -85,B 0,C 180,E1 -6429.249,E2 -6429.249} C_VEL
LIN {X 0,Y 488.727,Z 478.712,A -85,B 0,C 180,E1 -6432.52,E2 -6432.52} C_VEL
LIN {X 0,Y 488.694,Z 478.733,A -85,B 0,C 180,E1 -6435.976,E2 -6435.976} C_VEL
LIN {X 0,Y 488.71,Z 478.729,A -85,B 0,C 180,E1 -6438.585,E2 -6438.585} C_VEL
LIN {X 0,Y 488.672,Z 478.738,A -85,B 0,C 180,E1 -6441.8,E2 -6441.8} C_VEL
LIN {X 0,Y 488.72,Z 478.727,A -85,B 0,C 180,E1 -6445.051,E2 -6445.051} C_VEL
LIN {X 0,Y 488.697,Z 478.736,A -85,B 0,C 180,E1 -6448.045,E2 -6448.045} C_VEL
LIN {X 0,Y 488.724,Z 478.73,A -85,B 0,C 180,E1 -6450.73,E2 -6450.73} C_VEL
LIN {X 0,Y 488.757,Z 478.724,A -85,B 0,C 180,E1 -6453.529,E2 -6453.529} C_VEL
LIN {X 0,Y 488.682,Z 478.73,A -85,B 0,C 180,E1 -6456.255,E2 -6456.255} C_VEL
LIN {X 0,Y 488.736,Z 478.727,A -85,B 0,C 180,E1 -6459.176,E2 -6459.176} C_VEL
LIN {X 0,Y 488.749,Z 478.72,A -85,B 0,C 180,E1 -6461.628,E2 -6461.628} C_VEL
LIN {X 0,Y 488.752,Z 478.725,A -85,B 0,C 180,E1 -6465,E2 -6465} C_VEL
LIN {X 0,Y 488.798,Z 478.72,A -85,B 0,C 180,E1 -6468.388,E2 -6468.388} C_VEL
LIN {X 0,Y 488.808,Z 478.712,A -85,B 0,C 180,E1 -6471.734,E2 -6471.734} C_VEL
LIN {X 0,Y 488.86,Z 478.715,A -85,B 0,C 180,E1 -6474.225,E2 -6474.225} C_VEL
LIN {X 0,Y 488.953,Z 478.688,A -85,B 0,C 180,E1 -6477.529,E2 -6477.529} C_VEL
LIN {X 0,Y 488.946,Z 478.703,A -85,B 0,C 180,E1 -6480.824,E2 -6480.824} C_VEL
LIN {X 0,Y 488.953,Z 478.706,A -85,B 0,C 180,E1 -6482.472,E2 -6482.472} C_VEL
LIN {X 0,Y 488.847,Z 478.701,A -85,B 0,C 180,E1 -6485.776,E2 -6485.776} C_VEL
LIN {X 0,Y 488.809,Z 478.718,A -85,B 0,C 180,E1 -6488.267,E2 -6488.267} C_VEL
LIN {X 0,Y 488.796,Z 478.716,A -85,B 0,C 180,E1 -6491.613,E2 -6491.613} C_VEL
LIN {X 0,Y 488.753,Z 478.725,A -85,B 0,C 180,E1 -6495.001,E2 -6495.001} C_VEL
LIN {X 0,Y 488.747,Z 478.732,A -85,B 0,C 180,E1 -6498.443,E2 -6498.443} C_VEL
LIN {X 0,Y 488.7,Z 478.728,A -85,B 0,C 180,E1 -6501.071,E2 -6501.071} C_VEL
LIN {X 0,Y 488.686,Z 478.733,A -85,B 0,C 180,E1 -6503.746,E2 -6503.746} C_VEL
LIN {X 0,Y 488.792,Z 478.716,A -85,B 0,C 180,E1 -6506.946,E2 -6506.946} C_VEL
LIN {X 0,Y 488.703,Z 478.735,A -85,B 0,C 180,E1 -6510.364,E2 -6510.364} C_VEL
LIN {X 0,Y 488.73,Z 478.723,A -85,B 0,C 180,E1 -6513.485,E2 -6513.485} C_VEL
LIN {X 0,Y 488.683,Z 478.737,A -85,B 0,C 180,E1 -6516.356,E2 -6516.356} C_VEL
LIN {X 0,Y 488.733,Z 478.73,A -85,B 0,C 180,E1 -6519.252,E2 -6519.252} C_VEL
LIN {X 0,Y 488.706,Z 478.728,A -85,B 0,C 180,E1 -6521.601,E2 -6521.601} C_VEL
LIN {X 0,Y 488.708,Z 478.733,A -85,B 0,C 180,E1 -6524.802,E2 -6524.802} C_VEL
LIN {X 0,Y 488.692,Z 478.729,A -85,B 0,C 180,E1 -6527.476,E2 -6527.476} C_VEL
LIN {X 0,Y 488.73,Z 478.728,A -85,B 0,C 180,E1 -6529.677,E2 -6529.677} C_VEL
LIN {X 0,Y 488.676,Z 478.708,A -85,B 0,C 180,E1 -6532.842,E2 -6532.842} C_VEL
LIN {X 0,Y 488.73,Z 478.729,A -85,B 0,C 180,E1 -6535.888,E2 -6535.888} C_VEL
LIN {X 0,Y 488.692,Z 478.716,A -85,B 0,C 180,E1 -6538.821,E2 -6538.821} C_VEL
LIN {X 0,Y 488.769,Z 478.8,A -85,B 0,C 180,E1 -6541.345,E2 -6541.345} C_VEL
LIN {X 0,Y 490.934,Z 489.611,A -85,B 0,C 180,E1 -6543.655,E2 -6543.655} C_VEL
LIN {X 0,Y 490.942,Z 495.444,A -85,B 0,C 180,E1 -6544.794,E2 -6544.794} C_VEL
LIN {X 0,Y 490.338,Z 510.68,A -85,B 0,C 180,E1 -6547.678,E2 -6547.678} C_VEL
LIN {X 0,Y 489.797,Z 524.47,A -85,B 0,C 180,E1 -6550.251,E2 -6550.251} C_VEL
LIN {X 0,Y 491.797,Z 534.813,A -85,B 0,C 180,E1 -6550.521,E2 -6550.521} C_VEL
LIN {X 0,Y 493.461,Z 543.206,A -85,B 0,C 180,E1 -6550.715,E2 -6550.715} C_VEL
LIN {X 0,Y 492.534,Z 659.815,A -85,B 0,C 180,E1 -6552.457,E2 -6552.457} C_VEL
LIN {X 0,Y 492.25,Z 670.771,A -85,B 0,C 180,E1 -6552.714,E2 -6552.714} C_VEL
LIN {X 0,Y 491.951,Z 681.771,A -85,B 0,C 180,E1 -6553.078,E2 -6553.078} C_VEL
LIN {X 0,Y 491.606,Z 692.633,A -85,B 0,C 180,E1 -6553.547,E2 -6553.547} C_VEL
LIN {X 0,Y 491.236,Z 701.534,A -85,B 0,C 180,E1 -6554.014,E2 -6554.014} C_VEL
LIN {X 0,Y 490.824,Z 711.46,A -85,B 0,C 180,E1 -6554.64,E2 -6554.64} C_VEL
LIN {X 0,Y 490.311,Z 721.187,A -85,B 0,C 180,E1 -6555.367,E2 -6555.367} C_VEL
LIN {X 0,Y 489.833,Z 730.611,A -85,B 0,C 180,E1 -6556.2,E2 -6556.2} C_VEL
LIN {X 0,Y 489.441,Z 739.638,A -85,B 0,C 180,E1 -6557.14,E2 -6557.14} C_VEL
LIN {X 0,Y 489.042,Z 748.532,A -85,B 0,C 180,E1 -6558.231,E2 -6558.231} C_VEL
LIN {X 0,Y 488.737,Z 755.481,A -85,B 0,C 180,E1 -6559.226,E2 -6559.226} C_VEL
LIN {X 0,Y 488.485,Z 761.756,A -85,B 0,C 180,E1 -6560.268,E2 -6560.268} C_VEL
LIN {X 0,Y 488.306,Z 767.159,A -85,B 0,C 180,E1 -6561.308,E2 -6561.308} C_VEL
LIN {X 0,Y 488.095,Z 772.587,A -85,B 0,C 180,E1 -6562.554,E2 -6562.554} C_VEL
LIN {X 0,Y 488.012,Z 777.039,A -85,B 0,C 180,E1 -6563.803,E2 -6563.803} C_VEL
LIN {X 0,Y 487.961,Z 780.567,A -85,B 0,C 180,E1 -6565.043,E2 -6565.043} C_VEL
LIN {X 0,Y 487.908,Z 782.503,A -85,B 0,C 180,E1 -6565.87,E2 -6565.87} C_VEL
LIN {X 0,Y 487.906,Z 785.18,A -85,B 0,C 180,E1 -6567.523,E2 -6567.523} C_VEL
LIN {X 0,Y 487.831,Z 786.463,A -85,B 0,C 180,E1 -6569.175,E2 -6569.175} C_VEL
LIN {X 0,Y 487.817,Z 786.714,A -85,B 0,C 180,E1 -6570,E2 -6570} C_VEL
LIN {X 0,Y 487.887,Z 785.994,A -85,B 0,C 180,E1 -6571.651,E2 -6571.651} C_VEL
LIN {X 0,Y 487.906,Z 785.18,A -85,B 0,C 180,E1 -6572.477,E2 -6572.477} C_VEL
LIN {X 0,Y 487.908,Z 782.503,A -85,B 0,C 180,E1 -6574.13,E2 -6574.13} C_VEL
LIN {X 0,Y 488.013,Z 779.555,A -85,B 0,C 180,E1 -6575.371,E2 -6575.371} C_VEL
LIN {X 0,Y 488.043,Z 775.732,A -85,B 0,C 180,E1 -6576.615,E2 -6576.615} C_VEL
LIN {X 0,Y 488.171,Z 770.974,A -85,B 0,C 180,E1 -6577.861,E2 -6577.861} C_VEL
LIN {X 0,Y 488.41,Z 764.032,A -85,B 0,C 180,E1 -6579.316,E2 -6579.316} C_VEL
LIN {X 0,Y 488.69,Z 756.819,A -85,B 0,C 180,E1 -6580.565,E2 -6580.565} C_VEL
LIN {X 0,Y 488.985,Z 749.742,A -85,B 0,C 180,E1 -6581.608,E2 -6581.608} C_VEL
LIN {X 0,Y 489.359,Z 741.458,A -85,B 0,C 180,E1 -6582.651,E2 -6582.651} C_VEL
LIN {X 0,Y 489.761,Z 732.733,A -85,B 0,C 180,E1 -6583.59,E2 -6583.59} C_VEL
LIN {X 0,Y 490.19,Z 723.669,A -85,B 0,C 180,E1 -6584.425,E2 -6584.425} C_VEL
LIN {X 0,Y 490.666,Z 714.389,A -85,B 0,C 180,E1 -6585.153,E2 -6585.153} C_VEL
LIN {X 0,Y 491.102,Z 705.044,A -85,B 0,C 180,E1 -6585.777,E2 -6585.777} C_VEL
LIN {X 0,Y 491.501,Z 694.78,A -85,B 0,C 180,E1 -6586.35,E2 -6586.35} C_VEL
LIN {X 0,Y 491.889,Z 683.805,A -85,B 0,C 180,E1 -6586.844,E2 -6586.844} C_VEL
LIN {X 0,Y 492.21,Z 673.321,A -85,B 0,C 180,E1 -6587.212,E2 -6587.212} C_VEL
LIN {X 0,Y 492.507,Z 661.174,A -85,B 0,C 180,E1 -6587.518,E2 -6587.518} C_VEL
LIN {X 0,Y 492.816,Z 632.852,A -85,B 0,C 180,E1 -6587.962,E2 -6587.962} C_VEL
LIN {X 0,Y 493.465,Z 543.457,A -85,B 0,C 180,E1 -6589.281,E2 -6589.281} C_VEL
LIN {X 0,Y 489.799,Z 524.544,A -85,B 0,C 180,E1 -6589.744,E2 -6589.744} C_VEL
LIN {X 0,Y 490.348,Z 510.763,A -85,B 0,C 180,E1 -6592.322,E2 -6592.322} C_VEL
LIN {X 0,Y 490.948,Z 495.444,A -85,B 0,C 180,E1 -6595.205,E2 -6595.205} C_VEL
LIN {X 0,Y 491.033,Z 490.673,A -85,B 0,C 180,E1 -6596.13,E2 -6596.13} C_VEL
LIN {X 0,Y 489.063,Z 480.265,A -85,B 0,C 180,E1 -6598.308,E2 -6598.308} C_VEL
LIN {X 0,Y 488.741,Z 478.76,A -85,B 0,C 180,E1 -6598.697,E2 -6598.697} C_VEL
LIN {X 0,Y 488.704,Z 478.724,A -85,B 0,C 180,E1 -6601.954,E2 -6601.954} C_VEL
LIN {X 0,Y 488.722,Z 478.719,A -85,B 0,C 180,E1 -6604.947,E2 -6604.947} C_VEL
LIN {X 0,Y 488.677,Z 478.723,A -85,B 0,C 180,E1 -6608.199,E2 -6608.199} C_VEL
LIN {X 0,Y 488.716,Z 478.732,A -85,B 0,C 180,E1 -6611.414,E2 -6611.414} C_VEL
LIN {X 0,Y 488.698,Z 478.726,A -85,B 0,C 180,E1 -6614.023,E2 -6614.023} C_VEL
LIN {X 0,Y 488.68,Z 478.739,A -85,B 0,C 180,E1 -6617.176,E2 -6617.176} C_VEL
LIN {X 0,Y 488.728,Z 478.731,A -85,B 0,C 180,E1 -6619.676,E2 -6619.676} C_VEL
LIN {X 0,Y 488.674,Z 478.73,A -85,B 0,C 180,E1 -6622.277,E2 -6622.277} C_VEL
LIN {X 0,Y 488.723,Z 478.733,A -85,B 0,C 180,E1 -6625.051,E2 -6625.051} C_VEL
LIN {X 0,Y 488.699,Z 478.73,A -85,B 0,C 180,E1 -6628.045,E2 -6628.045} C_VEL
LIN {X 0,Y 488.717,Z 478.73,A -85,B 0,C 180,E1 -6630.729,E2 -6630.729} C_VEL
LIN {X 0,Y 488.76,Z 478.724,A -85,B 0,C 180,E1 -6633.528,E2 -6633.528} C_VEL
LIN {X 0,Y 488.686,Z 478.733,A -85,B 0,C 180,E1 -6636.254,E2 -6636.254} C_VEL
LIN {X 0,Y 488.738,Z 478.723,A -85,B 0,C 180,E1 -6639.175,E2 -6639.175} C_VEL
LIN {X 0,Y 488.751,Z 478.73,A -85,B 0,C 180,E1 -6641.627,E2 -6641.627} C_VEL
LIN {X 0,Y 488.753,Z 478.725,A -85,B 0,C 180,E1 -6644.999,E2 -6644.999} C_VEL
LIN {X 0,Y 488.796,Z 478.716,A -85,B 0,C 180,E1 -6648.387,E2 -6648.387} C_VEL
LIN {X 0,Y 488.809,Z 478.718,A -85,B 0,C 180,E1 -6651.733,E2 -6651.733} C_VEL
LIN {X 0,Y 488.847,Z 478.701,A -85,B 0,C 180,E1 -6654.224,E2 -6654.224} C_VEL
LIN {X 0,Y 488.953,Z 478.706,A -85,B 0,C 180,E1 -6657.528,E2 -6657.528} C_VEL
LIN {X 0,Y 488.946,Z 478.695,A -85,B 0,C 180,E1 -6660.823,E2 -6660.823} C_VEL
LIN {X 0,Y 488.952,Z 478.688,A -85,B 0,C 180,E1 -6662.471,E2 -6662.471} C_VEL
LIN {X 0,Y 488.846,Z 478.717,A -85,B 0,C 180,E1 -6665.775,E2 -6665.775} C_VEL
LIN {X 0,Y 488.808,Z 478.712,A -85,B 0,C 180,E1 -6668.266,E2 -6668.266} C_VEL
LIN {X 0,Y 488.798,Z 478.72,A -85,B 0,C 180,E1 -6671.612,E2 -6671.612} C_VEL
LIN {X 0,Y 488.752,Z 478.725,A -85,B 0,C 180,E1 -6675,E2 -6675} C_VEL
LIN {X 0,Y 488.745,Z 478.72,A -85,B 0,C 180,E1 -6678.442,E2 -6678.442} C_VEL
LIN {X 0,Y 488.697,Z 478.733,A -85,B 0,C 180,E1 -6681.071,E2 -6681.071} C_VEL
LIN {X 0,Y 488.682,Z 478.73,A -85,B 0,C 180,E1 -6683.745,E2 -6683.745} C_VEL
LIN {X 0,Y 488.789,Z 478.72,A -85,B 0,C 180,E1 -6686.945,E2 -6686.945} C_VEL
LIN {X 0,Y 488.709,Z 478.723,A -85,B 0,C 180,E1 -6690.365,E2 -6690.365} C_VEL
LIN {X 0,Y 488.727,Z 478.733,A -85,B 0,C 180,E1 -6693.485,E2 -6693.485} C_VEL
LIN {X 0,Y 488.68,Z 478.731,A -85,B 0,C 180,E1 -6696.356,E2 -6696.356} C_VEL
LIN {X 0,Y 488.693,Z 478.735,A -85,B 0,C 180,E1 -6699.254,E2 -6699.254} C_VEL
LIN {X 0,Y 488.727,Z 478.729,A -85,B 0,C 180,E1 -6702.521,E2 -6702.521} C_VEL
LIN {X 0,Y 488.694,Z 478.718,A -85,B 0,C 180,E1 -6705.976,E2 -6705.976} C_VEL
LIN {X 0,Y 488.722,Z 478.726,A -85,B 0,C 180,E1 -6708.587,E2 -6708.587} C_VEL
LIN {X 0,Y 488.741,Z 478.727,A -85,B 0,C 180,E1 -6710.941,E2 -6710.941} C_VEL
LIN {X 0,Y 488.678,Z 478.728,A -85,B 0,C 180,E1 -6713.869,E2 -6713.869} C_VEL
LIN {X 0,Y 488.733,Z 478.728,A -85,B 0,C 180,E1 -6716.878,E2 -6716.878} C_VEL
LIN {X 0,Y 488.728,Z 478.736,A -85,B 0,C 180,E1 -6719.782,E2 -6719.782} C_VEL
LIN {X 0,Y 488.786,Z 478.723,A -85,B 0,C 180,E1 -6723.057,E2 -6723.057} C_VEL
LIN {X 0,Y 488.738,Z 478.729,A -85,B 0,C 180,E1 -6724.359,E2 -6724.359} C_VEL
LIN {X 0,Y 488.094,Z 478.813,A -85,B 0,C 180,E1 -6725.047,E2 -6725.047} C_VEL
LIN {X 0,Y 485.227,Z 479.174,A -85,B 0,C 180,E1 -6726.163,E2 -6726.163} C_VEL
LIN {X 0,Y 482.781,Z 479.478,A -85,B 0,C 180,E1 -6727.063,E2 -6727.063} C_VEL
LIN {X 0,Y 481.722,Z 479.608,A -85,B 0,C 180,E1 -6727.758,E2 -6727.758} C_VEL
LIN {X 0,Y 481.633,Z 479.616,A -85,B 0,C 180,E1 -6727.994,E2 -6727.994} C_VEL
LIN {X 0,Y 481.701,Z 479.608,A -85,B 0,C 180,E1 -6730.393,E2 -6730.393} C_VEL
LIN {X 0,Y 481.687,Z 479.608,A -85,B 0,C 180,E1 -6733.034,E2 -6733.034} C_VEL
LIN {X 0,Y 481.686,Z 479.611,A -85,B 0,C 180,E1 -6735.639,E2 -6735.639} C_VEL
LIN {X 0,Y 481.747,Z 479.604,A -85,B 0,C 180,E1 -6738.215,E2 -6738.215} C_VEL
LIN {X 0,Y 481.759,Z 479.602,A -85,B 0,C 180,E1 -6741.612,E2 -6741.612} C_VEL
LIN {X 0,Y 481.812,Z 479.597,A -85,B 0,C 180,E1 -6744.14,E2 -6744.14} C_VEL
LIN {X 0,Y 481.925,Z 479.581,A -85,B 0,C 180,E1 -6747.493,E2 -6747.493} C_VEL
LIN {X 0,Y 481.902,Z 479.582,A -85,B 0,C 180,E1 -6750.836,E2 -6750.836} C_VEL
LIN {X 0,Y 481.925,Z 479.581,A -85,B 0,C 180,E1 -6752.507,E2 -6752.507} C_VEL
LIN {X 0,Y 481.812,Z 479.597,A -85,B 0,C 180,E1 -6755.86,E2 -6755.86} C_VEL
LIN {X 0,Y 481.759,Z 479.602,A -85,B 0,C 180,E1 -6758.388,E2 -6758.388} C_VEL
LIN {X 0,Y 481.747,Z 479.604,A -85,B 0,C 180,E1 -6761.785,E2 -6761.785} C_VEL
LIN {X 0,Y 481.738,Z 479.602,A -85,B 0,C 180,E1 -6765.224,E2 -6765.224} C_VEL
LIN {X 0,Y 481.708,Z 479.606,A -85,B 0,C 180,E1 -6768.721,E2 -6768.721} C_VEL
LIN {X 0,Y 481.642,Z 479.613,A -85,B 0,C 180,E1 -6771.394,E2 -6771.394} C_VEL
LIN {X 0,Y 481.672,Z 479.614,A -85,B 0,C 180,E1 -6774.113,E2 -6774.113} C_VEL
LIN {X 0,Y 481.741,Z 479.6,A -85,B 0,C 180,E1 -6777.139,E2 -6777.139} C_VEL
LIN {X 0,Y 481.682,Z 479.61,A -85,B 0,C 180,E1 -6779.74,E2 -6779.74} C_VEL
LIN {X 0,Y 481.667,Z 479.611,A -85,B 0,C 180,E1 -6782.674,E2 -6782.674} C_VEL
LIN {X 0,Y 481.636,Z 479.611,A -85,B 0,C 180,E1 -6785.709,E2 -6785.709} C_VEL
LIN {X 0,Y 481.712,Z 479.602,A -85,B 0,C 180,E1 -6789.354,E2 -6789.354} C_VEL
LIN {X 0,Y 481.667,Z 479.596,A -85,B 0,C 180,E1 -6792.157,E2 -6792.157} C_VEL
LIN {X 0,Y 481.652,Z 479.603,A -85,B 0,C 180,E1 -6794.457,E2 -6794.457} C_VEL
LIN {X 0,Y 481.681,Z 479.608,A -85,B 0,C 180,E1 -6796.845,E2 -6796.845} C_VEL
LIN {X 0,Y 481.668,Z 479.607,A -85,B 0,C 180,E1 -6800.059,E2 -6800.059} C_VEL
LIN {X 0,Y 481.62,Z 479.609,A -85,B 0,C 180,E1 -6803.253,E2 -6803.253} C_VEL
LIN {X 0,Y 481.7,Z 479.611,A -85,B 0,C 180,E1 -6806.33,E2 -6806.33} C_VEL
LIN {X 0,Y 481.649,Z 479.601,A -85,B 0,C 180,E1 -6809.416,E2 -6809.416} C_VEL
LIN {X 0,Y 481.693,Z 479.609,A -85,B 0,C 180,E1 -6812.168,E2 -6812.168} C_VEL
LIN {X 0,Y 481.708,Z 479.595,A -85,B 0,C 180,E1 -6814.97,E2 -6814.97} C_VEL
LIN {X 0,Y 481.64,Z 479.609,A -85,B 0,C 180,E1 -6817.705,E2 -6817.705} C_VEL
LIN {X 0,Y 481.698,Z 479.607,A -85,B 0,C 180,E1 -6820.393,E2 -6820.393} C_VEL
LIN {X 0,Y 481.682,Z 479.599,A -85,B 0,C 180,E1 -6823.034,E2 -6823.034} C_VEL
LIN {X 0,Y 481.679,Z 479.605,A -85,B 0,C 180,E1 -6825.639,E2 -6825.639} C_VEL
LIN {X 0,Y 481.742,Z 479.602,A -85,B 0,C 180,E1 -6828.215,E2 -6828.215} C_VEL
LIN {X 0,Y 481.754,Z 479.59,A -85,B 0,C 180,E1 -6831.612,E2 -6831.612} C_VEL
LIN {X 0,Y 481.819,Z 479.591,A -85,B 0,C 180,E1 -6834.14,E2 -6834.14} C_VEL
LIN {X 0,Y 481.919,Z 479.563,A -85,B 0,C 180,E1 -6837.493,E2 -6837.493} C_VEL
LIN {X 0,Y 481.897,Z 479.581,A -85,B 0,C 180,E1 -6840.836,E2 -6840.836} C_VEL
LIN {X 0,Y 481.92,Z 479.581,A -85,B 0,C 180,E1 -6842.508,E2 -6842.508} C_VEL
LIN {X 0,Y 481.808,Z 479.577,A -85,B 0,C 180,E1 -6845.861,E2 -6845.861} C_VEL
LIN {X 0,Y 481.755,Z 479.599,A -85,B 0,C 180,E1 -6848.389,E2 -6848.389} C_VEL
LIN {X 0,Y 481.742,Z 479.595,A -85,B 0,C 180,E1 -6851.785,E2 -6851.785} C_VEL
LIN {X 0,Y 481.734,Z 479.597,A -85,B 0,C 180,E1 -6855.225,E2 -6855.225} C_VEL
LIN {X 0,Y 481.704,Z 479.604,A -85,B 0,C 180,E1 -6858.722,E2 -6858.722} C_VEL
LIN {X 0,Y 481.639,Z 479.605,A -85,B 0,C 180,E1 -6861.395,E2 -6861.395} C_VEL
LIN {X 0,Y 481.67,Z 479.609,A -85,B 0,C 180,E1 -6864.114,E2 -6864.114} C_VEL
LIN {X 0,Y 481.745,Z 479.592,A -85,B 0,C 180,E1 -6867.141,E2 -6867.141} C_VEL
LIN {X 0,Y 481.672,Z 479.606,A -85,B 0,C 180,E1 -6869.742,E2 -6869.742} C_VEL
LIN {X 0,Y 481.667,Z 479.607,A -85,B 0,C 180,E1 -6872.675,E2 -6872.675} C_VEL
LIN {X 0,Y 481.637,Z 479.611,A -85,B 0,C 180,E1 -6875.71,E2 -6875.71} C_VEL
LIN {X 0,Y 481.706,Z 479.604,A -85,B 0,C 180,E1 -6879.354,E2 -6879.354} C_VEL
LIN {X 0,Y 481.644,Z 479.609,A -85,B 0,C 180,E1 -6882.161,E2 -6882.161} C_VEL
LIN {X 0,Y 481.657,Z 479.604,A -85,B 0,C 180,E1 -6885.544,E2 -6885.544} C_VEL
LIN {X 0,Y 481.659,Z 479.605,A -85,B 0,C 180,E1 -6888.087,E2 -6888.087} C_VEL
LIN {X 0,Y 481.669,Z 479.599,A -85,B 0,C 180,E1 -6891.142,E2 -6891.142} C_VEL
LIN {X 0,Y 481.661,Z 479.591,A -85,B 0,C 180,E1 -6894.797,E2 -6894.797} C_VEL
LIN {X 0,Y 481.671,Z 479.606,A -85,B 0,C 180,E1 -6897.327,E2 -6897.327} C_VEL
LIN {X 0,Y 481.704,Z 479.61,A -85,B 0,C 180,E1 -6900.948,E2 -6900.948} C_VEL
LIN {X 0,Y 481.727,Z 479.819,A -85,B 0,C 180,E1 -6901.152,E2 -6901.152} C_VEL
LIN {X 0,Y 484.096,Z 491.762,A -85,B 0,C 180,E1 -6903.719,E2 -6903.719} C_VEL
LIN {X 0,Y 483.885,Z 499.993,A -85,B 0,C 180,E1 -6905.319,E2 -6905.319} C_VEL
LIN {X 0,Y 483.226,Z 515.381,A -85,B 0,C 180,E1 -6908.276,E2 -6908.276} C_VEL
LIN {X 0,Y 482.833,Z 524.267,A -85,B 0,C 180,E1 -6909.954,E2 -6909.954} C_VEL
LIN {X 0,Y 484.758,Z 534.01,A -85,B 0,C 180,E1 -6910.217,E2 -6910.217} C_VEL
LIN {X 0,Y 486.782,Z 545.215,A -85,B 0,C 180,E1 -6910.474,E2 -6910.474} C_VEL
LIN {X 0,Y 485.757,Z 659.616,A -85,B 0,C 180,E1 -6912.204,E2 -6912.204} C_VEL
LIN {X 0,Y 485.466,Z 670.573,A -85,B 0,C 180,E1 -6912.465,E2 -6912.465} C_VEL
LIN {X 0,Y 485.16,Z 681.573,A -85,B 0,C 180,E1 -6912.834,E2 -6912.834} C_VEL
LIN {X 0,Y 484.792,Z 692.164,A -85,B 0,C 180,E1 -6913.295,E2 -6913.295} C_VEL
LIN {X 0,Y 484.38,Z 701.407,A -85,B 0,C 180,E1 -6913.786,E2 -6913.786} C_VEL
LIN {X 0,Y 483.945,Z 711.26,A -85,B 0,C 180,E1 -6914.416,E2 -6914.416} C_VEL
LIN {X 0,Y 483.393,Z 720.988,A -85,B 0,C 180,E1 -6915.153,E2 -6915.153} C_VEL
LIN {X 0,Y 482.917,Z 730.412,A -85,B 0,C 180,E1 -6915.999,E2 -6915.999} C_VEL
LIN {X 0,Y 482.474,Z 739.439,A -85,B 0,C 180,E1 -6916.951,E2 -6916.951} C_VEL
LIN {X 0,Y 482.063,Z 747.75,A -85,B 0,C 180,E1 -6917.978,E2 -6917.978} C_VEL
LIN {X 0,Y 481.719,Z 755.282,A -85,B 0,C 180,E1 -6919.067,E2 -6919.067} C_VEL
LIN {X 0,Y 481.439,Z 761.557,A -85,B 0,C 180,E1 -6920.124,E2 -6920.124} C_VEL
LIN {X 0,Y 481.227,Z 766.959,A -85,B 0,C 180,E1 -6921.179,E2 -6921.179} C_VEL
LIN {X 0,Y 481.019,Z 772.388,A -85,B 0,C 180,E1 -6922.444,E2 -6922.444} C_VEL
LIN {X 0,Y 480.997,Z 776.205,A -85,B 0,C 180,E1 -6923.501,E2 -6923.501} C_VEL
LIN {X 0,Y 480.892,Z 780.37,A -85,B 0,C 180,E1 -6924.97,E2 -6924.97} C_VEL
LIN {X 0,Y 480.812,Z 782.304,A -85,B 0,C 180,E1 -6925.809,E2 -6925.809} C_VEL
LIN {X 0,Y 480.82,Z 784.982,A -85,B 0,C 180,E1 -6927.487,E2 -6927.487} C_VEL
LIN {X 0,Y 480.757,Z 786.266,A -85,B 0,C 180,E1 -6929.162,E2 -6929.162} C_VEL
LIN {X 0,Y 480.741,Z 786.517,A -85,B 0,C 180,E1 -6930,E2 -6930} C_VEL
LIN {X 0,Y 480.789,Z 785.796,A -85,B 0,C 180,E1 -6931.675,E2 -6931.675} C_VEL
LIN {X 0,Y 480.82,Z 784.982,A -85,B 0,C 180,E1 -6932.513,E2 -6932.513} C_VEL
LIN {X 0,Y 480.812,Z 782.304,A -85,B 0,C 180,E1 -6934.191,E2 -6934.191} C_VEL
LIN {X 0,Y 480.926,Z 779.356,A -85,B 0,C 180,E1 -6935.45,E2 -6935.45} C_VEL
LIN {X 0,Y 480.962,Z 775.533,A -85,B 0,C 180,E1 -6936.713,E2 -6936.713} C_VEL
LIN {X 0,Y 481.098,Z 770.774,A -85,B 0,C 180,E1 -6937.977,E2 -6937.977} C_VEL
LIN {X 0,Y 481.373,Z 763.833,A -85,B 0,C 180,E1 -6939.453,E2 -6939.453} C_VEL
LIN {X 0,Y 481.661,Z 756.62,A -85,B 0,C 180,E1 -6940.721,E2 -6940.721} C_VEL
LIN {X 0,Y 481.963,Z 749.542,A -85,B 0,C 180,E1 -6941.779,E2 -6941.779} C_VEL
LIN {X 0,Y 482.372,Z 741.258,A -85,B 0,C 180,E1 -6942.837,E2 -6942.837} C_VEL
LIN {X 0,Y 482.814,Z 732.533,A -85,B 0,C 180,E1 -6943.789,E2 -6943.789} C_VEL
LIN {X 0,Y 483.254,Z 723.469,A -85,B 0,C 180,E1 -6944.636,E2 -6944.636} C_VEL
LIN {X 0,Y 483.789,Z 714.19,A -85,B 0,C 180,E1 -6945.374,E2 -6945.374} C_VEL
LIN {X 0,Y 484.255,Z 704.845,A -85,B 0,C 180,E1 -6946.006,E2 -6946.006} C_VEL
LIN {X 0,Y 484.703,Z 693.858,A -85,B 0,C 180,E1 -6946.622,E2 -6946.622} C_VEL
LIN {X 0,Y 485.085,Z 683.607,A -85,B 0,C 180,E1 -6947.087,E2 -6947.087} C_VEL
LIN {X 0,Y 485.44,Z 672.119,A -85,B 0,C 180,E1 -6947.49,E2 -6947.49} C_VEL
LIN {X 0,Y 485.737,Z 660.976,A -85,B 0,C 180,E1 -6947.77,E2 -6947.77} C_VEL
LIN {X 0,Y 486.102,Z 630.864,A -85,B 0,C 180,E1 -6948.246,E2 -6948.246} C_VEL
LIN {X 0,Y 486.651,Z 543.905,A -85,B 0,C 180,E1 -6949.552,E2 -6949.552} C_VEL
LIN {X 0,Y 482.853,Z 524.463,A -85,B 0,C 180,E1 -6950.031,E2 -6950.031} C_VEL
LIN {X 0,Y 482.912,Z 522.079,A -85,B 0,C 180,E1 -6950.443,E2 -6950.443} C_VEL
LIN {X 0,Y 483.554,Z 508.248,A -85,B 0,C 180,E1 -6953.105,E2 -6953.105} C_VEL
LIN {X 0,Y 484.169,Z 492.923,A -85,B 0,C 180,E1 -6956.045,E2 -6956.045} C_VEL
LIN {X 0,Y 482.791,Z 484.792,A -85,B 0,C 180,E1 -6957.763,E2 -6957.763} C_VEL
LIN {X 0,Y 481.699,Z 479.65,A -85,B 0,C 180,E1 -6958.927,E2 -6958.927} C_VEL
LIN {X 0,Y 481.657,Z 479.605,A -85,B 0,C 180,E1 -6962.189,E2 -6962.189} C_VEL
LIN {X 0,Y 481.687,Z 479.6,A -85,B 0,C 180,E1 -6964.681,E2 -6964.681} C_VEL
LIN {X 0,Y 481.652,Z 479.596,A -85,B 0,C 180,E1 -6968.006,E2 -6968.006} C_VEL
LIN {X 0,Y 481.66,Z 479.615,A -85,B 0,C 180,E1 -6971.04,E2 -6971.04} C_VEL
LIN {X 0,Y 481.655,Z 479.603,A -85,B 0,C 180,E1 -6974.358,E2 -6974.358} C_VEL
LIN {X 0,Y 481.628,Z 479.616,A -85,B 0,C 180,E1 -6976.852,E2 -6976.852} C_VEL
LIN {X 0,Y 481.683,Z 479.606,A -85,B 0,C 180,E1 -6980.06,E2 -6980.06} C_VEL
LIN {X 0,Y 481.624,Z 479.616,A -85,B 0,C 180,E1 -6983.253,E2 -6983.253} C_VEL
LIN {X 0,Y 481.704,Z 479.598,A -85,B 0,C 180,E1 -6986.329,E2 -6986.329} C_VEL
LIN {X 0,Y 481.645,Z 479.618,A -85,B 0,C 180,E1 -6989.416,E2 -6989.416} C_VEL
LIN {X 0,Y 481.695,Z 479.597,A -85,B 0,C 180,E1 -6992.167,E2 -6992.167} C_VEL
LIN {X 0,Y 481.711,Z 479.602,A -85,B 0,C 180,E1 -6994.969,E2 -6994.969} C_VEL
LIN {X 0,Y 481.643,Z 479.608,A -85,B 0,C 180,E1 -6997.704,E2 -6997.704} C_VEL
LIN {X 0,Y 481.7,Z 479.597,A -85,B 0,C 180,E1 -7000.392,E2 -7000.392} C_VEL
LIN {X 0,Y 481.684,Z 479.608,A -85,B 0,C 180,E1 -7003.033,E2 -7003.033} C_VEL
LIN {X 0,Y 481.68,Z 479.599,A -85,B 0,C 180,E1 -7005.638,E2 -7005.638} C_VEL
LIN {X 0,Y 481.742,Z 479.595,A -85,B 0,C 180,E1 -7008.215,E2 -7008.215} C_VEL
LIN {X 0,Y 481.755,Z 479.599,A -85,B 0,C 180,E1 -7011.611,E2 -7011.611} C_VEL
LIN {X 0,Y 481.808,Z 479.577,A -85,B 0,C 180,E1 -7014.139,E2 -7014.139} C_VEL
LIN {X 0,Y 481.919,Z 479.581,A -85,B 0,C 180,E1 -7017.492,E2 -7017.492} C_VEL
LIN {X 0,Y 481.897,Z 479.573,A -85,B 0,C 180,E1 -7020.835,E2 -7020.835} C_VEL
LIN {X 0,Y 481.919,Z 479.563,A -85,B 0,C 180,E1 -7022.507,E2 -7022.507} C_VEL
LIN {X 0,Y 481.807,Z 479.593,A -85,B 0,C 180,E1 -7025.86,E2 -7025.86} C_VEL
LIN {X 0,Y 481.754,Z 479.59,A -85,B 0,C 180,E1 -7028.388,E2 -7028.388} C_VEL
LIN {X 0,Y 481.742,Z 479.602,A -85,B 0,C 180,E1 -7031.785,E2 -7031.785} C_VEL
LIN {X 0,Y 481.732,Z 479.602,A -85,B 0,C 180,E1 -7035.224,E2 -7035.224} C_VEL
LIN {X 0,Y 481.702,Z 479.597,A -85,B 0,C 180,E1 -7038.722,E2 -7038.722} C_VEL
LIN {X 0,Y 481.636,Z 479.616,A -85,B 0,C 180,E1 -7041.395,E2 -7041.395} C_VEL
LIN {X 0,Y 481.667,Z 479.601,A -85,B 0,C 180,E1 -7044.113,E2 -7044.113} C_VEL
LIN {X 0,Y 481.742,Z 479.599,A -85,B 0,C 180,E1 -7047.141,E2 -7047.141} C_VEL
LIN {X 0,Y 481.679,Z 479.604,A -85,B 0,C 180,E1 -7049.741,E2 -7049.741} C_VEL
LIN {X 0,Y 481.664,Z 479.607,A -85,B 0,C 180,E1 -7052.674,E2 -7052.674} C_VEL
LIN {X 0,Y 481.634,Z 479.612,A -85,B 0,C 180,E1 -7055.709,E2 -7055.709} C_VEL
LIN {X 0,Y 481.662,Z 479.609,A -85,B 0,C 180,E1 -7058.859,E2 -7058.859} C_VEL
LIN {X 0,Y 481.665,Z 479.611,A -85,B 0,C 180,E1 -7062.158,E2 -7062.158} C_VEL
LIN {X 0,Y 481.652,Z 479.606,A -85,B 0,C 180,E1 -7064.457,E2 -7064.457} C_VEL
LIN {X 0,Y 481.681,Z 479.584,A -85,B 0,C 180,E1 -7066.846,E2 -7066.846} C_VEL
LIN {X 0,Y 481.706,Z 479.608,A -85,B 0,C 180,E1 -7070.064,E2 -7070.064} C_VEL
LIN {X 0,Y 481.624,Z 479.603,A -85,B 0,C 180,E1 -7073.376,E2 -7073.376} C_VEL
LIN {X 0,Y 481.703,Z 479.606,A -85,B 0,C 180,E1 -7076.33,E2 -7076.33} C_VEL
LIN {X 0,Y 481.653,Z 479.614,A -85,B 0,C 180,E1 -7079.416,E2 -7079.416} C_VEL
LIN {X 0,Y 481.696,Z 479.61,A -85,B 0,C 180,E1 -7082.169,E2 -7082.169} C_VEL
LIN {X 0,Y 481.713,Z 479.604,A -85,B 0,C 180,E1 -7084.97,E2 -7084.97} C_VEL
LIN {X 0,Y 481.633,Z 479.616,A -85,B 0,C 180,E1 -7087.994,E2 -7087.994} C_VEL
LIN {X 0,Y 480.965,Z 479.698,A -85,B 0,C 180,E1 -7088.692,E2 -7088.692} C_VEL
LIN {X 0,Y 478.136,Z 480.054,A -85,B 0,C 180,E1 -7089.826,E2 -7089.826} C_VEL
LIN {X 0,Y 475.752,Z 480.349,A -85,B 0,C 180,E1 -7090.74,E2 -7090.74} C_VEL
LIN {X 0,Y 474.732,Z 480.477,A -85,B 0,C 180,E1 -7091.446,E2 -7091.446} C_VEL
LIN {X 0,Y 474.651,Z 480.487,A -85,B 0,C 180,E1 -7091.685,E2 -7091.685} C_VEL
LIN {X 0,Y 474.696,Z 480.48,A -85,B 0,C 180,E1 -7094.545,E2 -7094.545} C_VEL
LIN {X 0,Y 474.7,Z 480.482,A -85,B 0,C 180,E1 -7098.038,E2 -7098.038} C_VEL
LIN {X 0,Y 474.724,Z 480.477,A -85,B 0,C 180,E1 -7101.487,E2 -7101.487} C_VEL
LIN {X 0,Y 474.775,Z 480.473,A -85,B 0,C 180,E1 -7104.052,E2 -7104.052} C_VEL
LIN {X 0,Y 474.891,Z 480.457,A -85,B 0,C 180,E1 -7107.455,E2 -7107.455} C_VEL
LIN {X 0,Y 474.909,Z 480.457,A -85,B 0,C 180,E1 -7110,E2 -7110} C_VEL
LIN {X 0,Y 474.891,Z 480.457,A -85,B 0,C 180,E1 -7112.545,E2 -7112.545} C_VEL
LIN {X 0,Y 474.775,Z 480.473,A -85,B 0,C 180,E1 -7115.947,E2 -7115.947} C_VEL
LIN {X 0,Y 474.724,Z 480.477,A -85,B 0,C 180,E1 -7118.513,E2 -7118.513} C_VEL
LIN {X 0,Y 474.7,Z 480.482,A -85,B 0,C 180,E1 -7121.962,E2 -7121.962} C_VEL
LIN {X 0,Y 474.696,Z 480.48,A -85,B 0,C 180,E1 -7125.455,E2 -7125.455} C_VEL
LIN {X 0,Y 474.66,Z 480.483,A -85,B 0,C 180,E1 -7129.01,E2 -7129.01} C_VEL
LIN {X 0,Y 474.586,Z 480.495,A -85,B 0,C 180,E1 -7131.728,E2 -7131.728} C_VEL
LIN {X 0,Y 474.654,Z 480.487,A -85,B 0,C 180,E1 -7134.493,E2 -7134.493} C_VEL
LIN {X 0,Y 474.693,Z 480.478,A -85,B 0,C 180,E1 -7137.338,E2 -7137.338} C_VEL
LIN {X 0,Y 474.604,Z 480.49,A -85,B 0,C 180,E1 -7140.811,E2 -7140.811} C_VEL
LIN {X 0,Y 474.632,Z 480.491,A -85,B 0,C 180,E1 -7143.984,E2 -7143.984} C_VEL
LIN {X 0,Y 474.568,Z 480.481,A -85,B 0,C 180,E1 -7146.9,E2 -7146.9} C_VEL
LIN {X 0,Y 474.648,Z 480.484,A -85,B 0,C 180,E1 -7149.651,E2 -7149.651} C_VEL
LIN {X 0,Y 474.644,Z 480.46,A -85,B 0,C 180,E1 -7152.93,E2 -7152.93} C_VEL
LIN {X 0,Y 474.61,Z 480.486,A -85,B 0,C 180,E1 -7155.896,E2 -7155.896} C_VEL
LIN {X 0,Y 474.623,Z 480.479,A -85,B 0,C 180,E1 -7159.04,E2 -7159.04} C_VEL
LIN {X 0,Y 474.602,Z 480.49,A -85,B 0,C 180,E1 -7161.704,E2 -7161.704} C_VEL
LIN {X 0,Y 474.621,Z 480.486,A -85,B 0,C 180,E1 -7164.726,E2 -7164.726} C_VEL
LIN {X 0,Y 474.629,Z 480.486,A -85,B 0,C 180,E1 -7167.788,E2 -7167.788} C_VEL
LIN {X 0,Y 474.623,Z 480.485,A -85,B 0,C 180,E1 -7170.883,E2 -7170.883} C_VEL
LIN {X 0,Y 474.657,Z 480.48,A -85,B 0,C 180,E1 -7173.629,E2 -7173.629} C_VEL
LIN {X 0,Y 474.626,Z 480.485,A -85,B 0,C 180,E1 -7176.641,E2 -7176.641} C_VEL
LIN {X 0,Y 474.647,Z 480.486,A -85,B 0,C 180,E1 -7180.09,E2 -7180.09} C_VEL
LIN {X 0,Y 474.641,Z 480.477,A -85,B 0,C 180,E1 -7182.775,E2 -7182.775} C_VEL
LIN {X 0,Y 474.638,Z 480.482,A -85,B 0,C 180,E1 -7185.421,E2 -7185.421} C_VEL
LIN {X 0,Y 474.695,Z 480.478,A -85,B 0,C 180,E1 -7188.038,E2 -7188.038} C_VEL
LIN {X 0,Y 474.719,Z 480.466,A -85,B 0,C 180,E1 -7191.487,E2 -7191.487} C_VEL
LIN {X 0,Y 474.779,Z 480.467,A -85,B 0,C 180,E1 -7194.053,E2 -7194.053} C_VEL
LIN {X 0,Y 474.886,Z 480.439,A -85,B 0,C 180,E1 -7197.456,E2 -7197.456} C_VEL
LIN {X 0,Y 474.849,Z 480.459,A -85,B 0,C 180,E1 -7200.848,E2 -7200.848} C_VEL
LIN {X 0,Y 474.886,Z 480.457,A -85,B 0,C 180,E1 -7202.545,E2 -7202.545} C_VEL
LIN {X 0,Y 474.77,Z 480.454,A -85,B 0,C 180,E1 -7205.948,E2 -7205.948} C_VEL
LIN {X 0,Y 474.72,Z 480.477,A -85,B 0,C 180,E1 -7208.514,E2 -7208.514} C_VEL
LIN {X 0,Y 474.695,Z 480.474,A -85,B 0,C 180,E1 -7211.963,E2 -7211.963} C_VEL
LIN {X 0,Y 474.691,Z 480.474,A -85,B 0,C 180,E1 -7215.456,E2 -7215.456} C_VEL
LIN {X 0,Y 474.658,Z 480.477,A -85,B 0,C 180,E1 -7219.011,E2 -7219.011} C_VEL
LIN {X 0,Y 474.582,Z 480.483,A -85,B 0,C 180,E1 -7221.73,E2 -7221.73} C_VEL
LIN {X 0,Y 474.652,Z 480.488,A -85,B 0,C 180,E1 -7224.494,E2 -7224.494} C_VEL
LIN {X 0,Y 474.692,Z 480.469,A -85,B 0,C 180,E1 -7227.339,E2 -7227.339} C_VEL
LIN {X 0,Y 474.599,Z 480.492,A -85,B 0,C 180,E1 -7230.811,E2 -7230.811} C_VEL
LIN {X 0,Y 474.632,Z 480.479,A -85,B 0,C 180,E1 -7233.985,E2 -7233.985} C_VEL
LIN {X 0,Y 474.57,Z 480.492,A -85,B 0,C 180,E1 -7236.901,E2 -7236.901} C_VEL
LIN {X 0,Y 474.643,Z 480.483,A -85,B 0,C 180,E1 -7239.651,E2 -7239.651} C_VEL
LIN {X 0,Y 474.602,Z 480.495,A -85,B 0,C 180,E1 -7242.936,E2 -7242.936} C_VEL
LIN {X 0,Y 474.611,Z 480.481,A -85,B 0,C 180,E1 -7245.897,E2 -7245.897} C_VEL
LIN {X 0,Y 474.629,Z 480.49,A -85,B 0,C 180,E1 -7249.041,E2 -7249.041} C_VEL
LIN {X 0,Y 474.607,Z 480.474,A -85,B 0,C 180,E1 -7251.705,E2 -7251.705} C_VEL
LIN {X 0,Y 474.623,Z 480.466,A -85,B 0,C 180,E1 -7254.726,E2 -7254.726} C_VEL
LIN {X 0,Y 474.636,Z 480.479,A -85,B 0,C 180,E1 -7257.789,E2 -7257.789} C_VEL
LIN {X 0,Y 474.696,Z 480.608,A -85,B 0,C 180,E1 -7260.87,E2 -7260.87} C_VEL
LIN {X 0,Y 477.118,Z 492.753,A -85,B 0,C 180,E1 -7263.54,E2 -7263.54} C_VEL
LIN {X 0,Y 477.093,Z 498.633,A -85,B 0,C 180,E1 -7264.711,E2 -7264.711} C_VEL
LIN {X 0,Y 476.378,Z 513.794,A -85,B 0,C 180,E1 -7267.674,E2 -7267.674} C_VEL
LIN {X 0,Y 475.9,Z 523.968,A -85,B 0,C 180,E1 -7269.637,E2 -7269.637} C_VEL
LIN {X 0,Y 476.719,Z 528.358,A -85,B 0,C 180,E1 -7269.784,E2 -7269.784} C_VEL
LIN {X 0,Y 480.084,Z 545.265,A -85,B 0,C 180,E1 -7270.194,E2 -7270.194} C_VEL
LIN {X 0,Y 479.016,Z 659.419,A -85,B 0,C 180,E1 -7271.945,E2 -7271.945} C_VEL
LIN {X 0,Y 478.702,Z 669.913,A -85,B 0,C 180,E1 -7272.195,E2 -7272.195} C_VEL
LIN {X 0,Y 478.365,Z 681.078,A -85,B 0,C 180,E1 -7272.571,E2 -7272.571} C_VEL
LIN {X 0,Y 478.011,Z 691.26,A -85,B 0,C 180,E1 -7273.015,E2 -7273.015} C_VEL
LIN {X 0,Y 477.537,Z 701.41,A -85,B 0,C 180,E1 -7273.56,E2 -7273.56} C_VEL
LIN {X 0,Y 477.061,Z 711.061,A -85,B 0,C 180,E1 -7274.185,E2 -7274.185} C_VEL
LIN {X 0,Y 476.508,Z 720.789,A -85,B 0,C 180,E1 -7274.933,E2 -7274.933} C_VEL
LIN {X 0,Y 476.022,Z 730.214,A -85,B 0,C 180,E1 -7275.792,E2 -7275.792} C_VEL
LIN {X 0,Y 475.492,Z 739.239,A -85,B 0,C 180,E1 -7276.756,E2 -7276.756} C_VEL
LIN {X 0,Y 475.153,Z 746.369,A -85,B 0,C 180,E1 -7277.637,E2 -7277.637} C_VEL
LIN {X 0,Y 474.808,Z 753.746,A -85,B 0,C 180,E1 -7278.69,E2 -7278.69} C_VEL
LIN {X 0,Y 474.379,Z 761.357,A -85,B 0,C 180,E1 -7279.975,E2 -7279.975} C_VEL
LIN {X 0,Y 474.169,Z 766.76,A -85,B 0,C 180,E1 -7281.047,E2 -7281.047} C_VEL
LIN {X 0,Y 473.964,Z 772.19,A -85,B 0,C 180,E1 -7282.331,E2 -7282.331} C_VEL
LIN {X 0,Y 473.915,Z 776.321,A -85,B 0,C 180,E1 -7283.509,E2 -7283.509} C_VEL
LIN {X 0,Y 473.823,Z 780.172,A -85,B 0,C 180,E1 -7284.894,E2 -7284.894} C_VEL
LIN {X 0,Y 473.721,Z 782.106,A -85,B 0,C 180,E1 -7285.746,E2 -7285.746} C_VEL
LIN {X 0,Y 473.738,Z 784.784,A -85,B 0,C 180,E1 -7287.449,E2 -7287.449} C_VEL
LIN {X 0,Y 473.686,Z 786.069,A -85,B 0,C 180,E1 -7289.15,E2 -7289.15} C_VEL
LIN {X 0,Y 473.668,Z 786.32,A -85,B 0,C 180,E1 -7290,E2 -7290} C_VEL
LIN {X 0,Y 473.695,Z 785.598,A -85,B 0,C 180,E1 -7291.7,E2 -7291.7} C_VEL
LIN {X 0,Y 473.738,Z 784.784,A -85,B 0,C 180,E1 -7292.551,E2 -7292.551} C_VEL
LIN {X 0,Y 473.721,Z 782.106,A -85,B 0,C 180,E1 -7294.254,E2 -7294.254} C_VEL
LIN {X 0,Y 473.84,Z 779.157,A -85,B 0,C 180,E1 -7295.532,E2 -7295.532} C_VEL
LIN {X 0,Y 473.893,Z 775.335,A -85,B 0,C 180,E1 -7296.814,E2 -7296.814} C_VEL
LIN {X 0,Y 474.039,Z 770.576,A -85,B 0,C 180,E1 -7298.097,E2 -7298.097} C_VEL
LIN {X 0,Y 474.324,Z 763.634,A -85,B 0,C 180,E1 -7299.595,E2 -7299.595} C_VEL
LIN {X 0,Y 474.569,Z 757.758,A -85,B 0,C 180,E1 -7300.668,E2 -7300.668} C_VEL
LIN {X 0,Y 474.925,Z 750.906,A -85,B 0,C 180,E1 -7301.74,E2 -7301.74} C_VEL
LIN {X 0,Y 475.312,Z 742.879,A -85,B 0,C 180,E1 -7302.814,E2 -7302.814} C_VEL
LIN {X 0,Y 475.816,Z 733.394,A -85,B 0,C 180,E1 -7303.887,E2 -7303.887} C_VEL
LIN {X 0,Y 476.298,Z 724.512,A -85,B 0,C 180,E1 -7304.745,E2 -7304.745} C_VEL
LIN {X 0,Y 476.841,Z 715.457,A -85,B 0,C 180,E1 -7305.494,E2 -7305.494} C_VEL
LIN {X 0,Y 477.406,Z 704.646,A -85,B 0,C 180,E1 -7306.242,E2 -7306.242} C_VEL
LIN {X 0,Y 477.855,Z 694.561,A -85,B 0,C 180,E1 -7306.822,E2 -7306.822} C_VEL
LIN {X 0,Y 478.285,Z 683.408,A -85,B 0,C 180,E1 -7307.338,E2 -7307.338} C_VEL
LIN {X 0,Y 478.679,Z 671.921,A -85,B 0,C 180,E1 -7307.745,E2 -7307.745} C_VEL
LIN {X 0,Y 478.983,Z 660.778,A -85,B 0,C 180,E1 -7308.029,E2 -7308.029} C_VEL
LIN {X 0,Y 479.342,Z 632.456,A -85,B 0,C 180,E1 -7308.485,E2 -7308.485} C_VEL
LIN {X 0,Y 480.036,Z 545.28,A -85,B 0,C 180,E1 -7309.808,E2 -7309.808} C_VEL
LIN {X 0,Y 475.934,Z 524.26,A -85,B 0,C 180,E1 -7310.335,E2 -7310.335} C_VEL
LIN {X 0,Y 475.95,Z 521.872,A -85,B 0,C 180,E1 -7310.756,E2 -7310.756} C_VEL
LIN {X 0,Y 476.666,Z 508.087,A -85,B 0,C 180,E1 -7313.458,E2 -7313.458} C_VEL
LIN {X 0,Y 477.216,Z 493.936,A -85,B 0,C 180,E1 -7316.219,E2 -7316.219} C_VEL
LIN {X 0,Y 475.28,Z 483.454,A -85,B 0,C 180,E1 -7318.481,E2 -7318.481} C_VEL
LIN {X 0,Y 474.684,Z 480.509,A -85,B 0,C 180,E1 -7319.195,E2 -7319.195} C_VEL
LIN {X 0,Y 474.615,Z 480.484,A -85,B 0,C 180,E1 -7322.43,E2 -7322.43} C_VEL
LIN {X 0,Y 474.612,Z 480.464,A -85,B 0,C 180,E1 -7325.468,E2 -7325.468} C_VEL
LIN {X 0,Y 474.609,Z 480.475,A -85,B 0,C 180,E1 -7328.456,E2 -7328.456} C_VEL
LIN {X 0,Y 474.629,Z 480.49,A -85,B 0,C 180,E1 -7330.959,E2 -7330.959} C_VEL
LIN {X 0,Y 474.611,Z 480.48,A -85,B 0,C 180,E1 -7334.103,E2 -7334.103} C_VEL
LIN {X 0,Y 474.602,Z 480.494,A -85,B 0,C 180,E1 -7337.064,E2 -7337.064} C_VEL
LIN {X 0,Y 474.643,Z 480.483,A -85,B 0,C 180,E1 -7340.349,E2 -7340.349} C_VEL
LIN {X 0,Y 474.588,Z 480.493,A -85,B 0,C 180,E1 -7343.676,E2 -7343.676} C_VEL
LIN {X 0,Y 474.637,Z 480.48,A -85,B 0,C 180,E1 -7346.779,E2 -7346.779} C_VEL
LIN {X 0,Y 474.599,Z 480.49,A -85,B 0,C 180,E1 -7349.769,E2 -7349.769} C_VEL
LIN {X 0,Y 474.708,Z 480.467,A -85,B 0,C 180,E1 -7352.68,E2 -7352.68} C_VEL
LIN {X 0,Y 474.652,Z 480.488,A -85,B 0,C 180,E1 -7355.506,E2 -7355.506} C_VEL
LIN {X 0,Y 474.663,Z 480.475,A -85,B 0,C 180,E1 -7359.185,E2 -7359.185} C_VEL
LIN {X 0,Y 474.649,Z 480.484,A -85,B 0,C 180,E1 -7361.884,E2 -7361.884} C_VEL
LIN {X 0,Y 474.691,Z 480.474,A -85,B 0,C 180,E1 -7364.544,E2 -7364.544} C_VEL
LIN {X 0,Y 474.695,Z 480.474,A -85,B 0,C 180,E1 -7368.037,E2 -7368.037} C_VEL
LIN {X 0,Y 474.72,Z 480.477,A -85,B 0,C 180,E1 -7371.486,E2 -7371.486} C_VEL
LIN {X 0,Y 474.77,Z 480.454,A -85,B 0,C 180,E1 -7374.052,E2 -7374.052} C_VEL
LIN {X 0,Y 474.886,Z 480.457,A -85,B 0,C 180,E1 -7377.455,E2 -7377.455} C_VEL
LIN {X 0,Y 474.849,Z 480.451,A -85,B 0,C 180,E1 -7380.848,E2 -7380.848} C_VEL
LIN {X 0,Y 474.886,Z 480.439,A -85,B 0,C 180,E1 -7382.544,E2 -7382.544} C_VEL
LIN {X 0,Y 474.769,Z 480.468,A -85,B 0,C 180,E1 -7385.947,E2 -7385.947} C_VEL
LIN {X 0,Y 474.719,Z 480.466,A -85,B 0,C 180,E1 -7388.513,E2 -7388.513} C_VEL
LIN {X 0,Y 474.695,Z 480.478,A -85,B 0,C 180,E1 -7391.962,E2 -7391.962} C_VEL
LIN {X 0,Y 474.69,Z 480.48,A -85,B 0,C 180,E1 -7395.456,E2 -7395.456} C_VEL
LIN {X 0,Y 474.656,Z 480.476,A -85,B 0,C 180,E1 -7399.01,E2 -7399.01} C_VEL
LIN {X 0,Y 474.579,Z 480.494,A -85,B 0,C 180,E1 -7401.729,E2 -7401.729} C_VEL
LIN {X 0,Y 474.649,Z 480.472,A -85,B 0,C 180,E1 -7404.493,E2 -7404.493} C_VEL
LIN {X 0,Y 474.689,Z 480.48,A -85,B 0,C 180,E1 -7407.339,E2 -7407.339} C_VEL
LIN {X 0,Y 474.6,Z 480.479,A -85,B 0,C 180,E1 -7410.811,E2 -7410.811} C_VEL
LIN {X 0,Y 474.629,Z 480.487,A -85,B 0,C 180,E1 -7413.984,E2 -7413.984} C_VEL
LIN {X 0,Y 474.566,Z 480.488,A -85,B 0,C 180,E1 -7416.9,E2 -7416.9} C_VEL
LIN {X 0,Y 474.619,Z 480.49,A -85,B 0,C 180,E1 -7419.648,E2 -7419.648} C_VEL
LIN {X 0,Y 474.644,Z 480.483,A -85,B 0,C 180,E1 -7422.93,E2 -7422.93} C_VEL
LIN {X 0,Y 474.61,Z 480.471,A -85,B 0,C 180,E1 -7425.897,E2 -7425.897} C_VEL
LIN {X 0,Y 474.64,Z 480.48,A -85,B 0,C 180,E1 -7429.038,E2 -7429.038} C_VEL
LIN {X 0,Y 474.612,Z 480.486,A -85,B 0,C 180,E1 -7431.703,E2 -7431.703} C_VEL
LIN {X 0,Y 474.623,Z 480.483,A -85,B 0,C 180,E1 -7434.726,E2 -7434.726} C_VEL
LIN {X 0,Y 474.632,Z 480.491,A -85,B 0,C 180,E1 -7437.788,E2 -7437.788} C_VEL
LIN {X 0,Y 474.626,Z 480.486,A -85,B 0,C 180,E1 -7440.883,E2 -7440.883} C_VEL
LIN {X 0,Y 474.655,Z 480.487,A -85,B 0,C 180,E1 -7443.629,E2 -7443.629} C_VEL
LIN {X 0,Y 474.631,Z 480.486,A -85,B 0,C 180,E1 -7446.641,E2 -7446.641} C_VEL
LIN {X 0,Y 474.65,Z 480.488,A -85,B 0,C 180,E1 -7450.09,E2 -7450.09} C_VEL
LIN {X 0,Y 474.651,Z 480.487,A -85,B 0,C 180,E1 -7451.685,E2 -7451.685} C_VEL
LIN {X 0,Y 473.989,Z 480.573,A -85,B 0,C 180,E1 -7452.394,E2 -7452.394} C_VEL
LIN {X 0,Y 471.137,Z 480.928,A -85,B 0,C 180,E1 -7453.546,E2 -7453.546} C_VEL
LIN {X 0,Y 468.72,Z 481.226,A -85,B 0,C 180,E1 -7454.474,E2 -7454.474} C_VEL
LIN {X 0,Y 467.679,Z 481.354,A -85,B 0,C 180,E1 -7455.191,E2 -7455.191} C_VEL
LIN {X 0,Y 467.592,Z 481.364,A -85,B 0,C 180,E1 -7455.434,E2 -7455.434} C_VEL
LIN {X 0,Y 467.649,Z 481.357,A -85,B 0,C 180,E1 -7458.734,E2 -7458.734} C_VEL
LIN {X 0,Y 467.745,Z 481.348,A -85,B 0,C 180,E1 -7462.228,E2 -7462.228} C_VEL
LIN {X 0,Y 467.721,Z 481.348,A -85,B 0,C 180,E1 -7464.828,E2 -7464.828} C_VEL
LIN {X 0,Y 467.857,Z 481.333,A -85,B 0,C 180,E1 -7467.417,E2 -7467.417} C_VEL
LIN {X 0,Y 467.879,Z 481.333,A -85,B 0,C 180,E1 -7470,E2 -7470} C_VEL
LIN {X 0,Y 467.857,Z 481.333,A -85,B 0,C 180,E1 -7472.583,E2 -7472.583} C_VEL
LIN {X 0,Y 467.74,Z 481.349,A -85,B 0,C 180,E1 -7476.037,E2 -7476.037} C_VEL
LIN {X 0,Y 467.678,Z 481.354,A -85,B 0,C 180,E1 -7478.643,E2 -7478.643} C_VEL
LIN {X 0,Y 467.652,Z 481.36,A -85,B 0,C 180,E1 -7482.145,E2 -7482.145} C_VEL
LIN {X 0,Y 467.635,Z 481.361,A -85,B 0,C 180,E1 -7485.695,E2 -7485.695} C_VEL
LIN {X 0,Y 467.613,Z 481.362,A -85,B 0,C 180,E1 -7488.764,E2 -7488.764} C_VEL
LIN {X 0,Y 467.576,Z 481.365,A -85,B 0,C 180,E1 -7491.268,E2 -7491.268} C_VEL
LIN {X 0,Y 467.569,Z 481.37,A -85,B 0,C 180,E1 -7493.943,E2 -7493.943} C_VEL
LIN {X 0,Y 467.611,Z 481.362,A -85,B 0,C 180,E1 -7496.8,E2 -7496.8} C_VEL
LIN {X 0,Y 467.582,Z 481.367,A -85,B 0,C 180,E1 -7499.735,E2 -7499.735} C_VEL
LIN {X 0,Y 467.577,Z 481.366,A -85,B 0,C 180,E1 -7502.758,E2 -7502.758} C_VEL
LIN {X 0,Y 467.55,Z 481.361,A -85,B 0,C 180,E1 -7505.889,E2 -7505.889} C_VEL
LIN {X 0,Y 467.611,Z 481.359,A -85,B 0,C 180,E1 -7509.141,E2 -7509.141} C_VEL
LIN {X 0,Y 467.611,Z 481.338,A -85,B 0,C 180,E1 -7512.571,E2 -7512.571} C_VEL
LIN {X 0,Y 467.566,Z 481.368,A -85,B 0,C 180,E1 -7516.176,E2 -7516.176} C_VEL
LIN {X 0,Y 467.575,Z 481.359,A -85,B 0,C 180,E1 -7518.722,E2 -7518.722} C_VEL
LIN {X 0,Y 467.557,Z 481.37,A -85,B 0,C 180,E1 -7521.955,E2 -7521.955} C_VEL
LIN {X 0,Y 467.559,Z 481.363,A -85,B 0,C 180,E1 -7525.168,E2 -7525.168} C_VEL
LIN {X 0,Y 467.576,Z 481.363,A -85,B 0,C 180,E1 -7528.26,E2 -7528.26} C_VEL
LIN {X 0,Y 467.573,Z 481.362,A -85,B 0,C 180,E1 -7531.251,E2 -7531.251} C_VEL
LIN {X 0,Y 467.602,Z 481.362,A -85,B 0,C 180,E1 -7534.16,E2 -7534.16} C_VEL
LIN {X 0,Y 467.567,Z 481.362,A -85,B 0,C 180,E1 -7536.996,E2 -7536.996} C_VEL
LIN {X 0,Y 467.614,Z 481.359,A -85,B 0,C 180,E1 -7539.777,E2 -7539.777} C_VEL
LIN {X 0,Y 467.599,Z 481.353,A -85,B 0,C 180,E1 -7542.507,E2 -7542.507} C_VEL
LIN {X 0,Y 467.596,Z 481.36,A -85,B 0,C 180,E1 -7545.197,E2 -7545.197} C_VEL
LIN {X 0,Y 467.647,Z 481.354,A -85,B 0,C 180,E1 -7547.855,E2 -7547.855} C_VEL
LIN {X 0,Y 467.673,Z 481.343,A -85,B 0,C 180,E1 -7551.358,E2 -7551.358} C_VEL
LIN {X 0,Y 467.742,Z 481.343,A -85,B 0,C 180,E1 -7553.963,E2 -7553.963} C_VEL
LIN {X 0,Y 467.851,Z 481.315,A -85,B 0,C 180,E1 -7557.417,E2 -7557.417} C_VEL
LIN {X 0,Y 467.873,Z 481.321,A -85,B 0,C 180,E1 -7560,E2 -7560} C_VEL
LIN {X 0,Y 467.851,Z 481.332,A -85,B 0,C 180,E1 -7562.583,E2 -7562.583} C_VEL
LIN {X 0,Y 467.735,Z 481.33,A -85,B 0,C 180,E1 -7566.038,E2 -7566.038} C_VEL
LIN {X 0,Y 467.673,Z 481.357,A -85,B 0,C 180,E1 -7568.643,E2 -7568.643} C_VEL
LIN {X 0,Y 467.647,Z 481.353,A -85,B 0,C 180,E1 -7572.146,E2 -7572.146} C_VEL
LIN {X 0,Y 467.631,Z 481.353,A -85,B 0,C 180,E1 -7575.696,E2 -7575.696} C_VEL
LIN {X 0,Y 467.61,Z 481.358,A -85,B 0,C 180,E1 -7578.765,E2 -7578.765} C_VEL
LIN {X 0,Y 467.573,Z 481.357,A -85,B 0,C 180,E1 -7581.269,E2 -7581.269} C_VEL
LIN {X 0,Y 467.566,Z 481.365,A -85,B 0,C 180,E1 -7583.944,E2 -7583.944} C_VEL
LIN {X 0,Y 467.621,Z 481.352,A -85,B 0,C 180,E1 -7586.8,E2 -7586.8} C_VEL
LIN {X 0,Y 467.548,Z 481.366,A -85,B 0,C 180,E1 -7589.739,E2 -7589.739} C_VEL
LIN {X 0,Y 467.578,Z 481.36,A -85,B 0,C 180,E1 -7592.759,E2 -7592.759} C_VEL
LIN {X 0,Y 467.551,Z 481.366,A -85,B 0,C 180,E1 -7595.89,E2 -7595.89} C_VEL
LIN {X 0,Y 467.608,Z 481.363,A -85,B 0,C 180,E1 -7599.142,E2 -7599.142} C_VEL
LIN {X 0,Y 467.582,Z 481.364,A -85,B 0,C 180,E1 -7602.568,E2 -7602.568} C_VEL
LIN {X 0,Y 467.567,Z 481.362,A -85,B 0,C 180,E1 -7605.054,E2 -7605.054} C_VEL
LIN {X 0,Y 467.586,Z 481.358,A -85,B 0,C 180,E1 -7607.441,E2 -7607.441} C_VEL
LIN {X 0,Y 467.58,Z 481.357,A -85,B 0,C 180,E1 -7610.856,E2 -7610.856} C_VEL
LIN {X 0,Y 467.558,Z 481.336,A -85,B 0,C 180,E1 -7614.262,E2 -7614.262} C_VEL
LIN {X 0,Y 467.581,Z 481.361,A -85,B 0,C 180,E1 -7617.322,E2 -7617.322} C_VEL
LIN {X 0,Y 467.633,Z 481.544,A -85,B 0,C 180,E1 -7620.624,E2 -7620.624} C_VEL
LIN {X 0,Y 469.877,Z 492.578,A -85,B 0,C 180,E1 -7623.1,E2 -7623.1} C_VEL
LIN {X 0,Y 470.319,Z 496.95,A -85,B 0,C 180,E1 -7624.017,E2 -7624.017} C_VEL
LIN {X 0,Y 469.574,Z 511.272,A -85,B 0,C 180,E1 -7626.867,E2 -7626.867} C_VEL
LIN {X 0,Y 468.976,Z 523.917,A -85,B 0,C 180,E1 -7629.339,E2 -7629.339} C_VEL
LIN {X 0,Y 473.3,Z 545.736,A -85,B 0,C 180,E1 -7629.908,E2 -7629.908} C_VEL
LIN {X 0,Y 472.317,Z 656.501,A -85,B 0,C 180,E1 -7631.624,E2 -7631.624} C_VEL
LIN {X 0,Y 471.996,Z 668.712,A -85,B 0,C 180,E1 -7631.903,E2 -7631.903} C_VEL
LIN {X 0,Y 471.614,Z 679.532,A -85,B 0,C 180,E1 -7632.258,E2 -7632.258} C_VEL
LIN {X 0,Y 471.221,Z 691.062,A -85,B 0,C 180,E1 -7632.763,E2 -7632.763} C_VEL
LIN {X 0,Y 470.705,Z 701.396,A -85,B 0,C 180,E1 -7633.326,E2 -7633.326} C_VEL
LIN {X 0,Y 470.213,Z 710.862,A -85,B 0,C 180,E1 -7633.948,E2 -7633.948} C_VEL
LIN {X 0,Y 469.631,Z 720.59,A -85,B 0,C 180,E1 -7634.707,E2 -7634.707} C_VEL
LIN {X 0,Y 469.084,Z 730.014,A -85,B 0,C 180,E1 -7635.577,E2 -7635.577} C_VEL
LIN {X 0,Y 468.526,Z 739.039,A -85,B 0,C 180,E1 -7636.556,E2 -7636.556} C_VEL
LIN {X 0,Y 468.136,Z 746.803,A -85,B 0,C 180,E1 -7637.538,E2 -7637.538} C_VEL
LIN {X 0,Y 467.81,Z 753.546,A -85,B 0,C 180,E1 -7638.518,E2 -7638.518} C_VEL
LIN {X 0,Y 467.341,Z 761.158,A -85,B 0,C 180,E1 -7639.823,E2 -7639.823} C_VEL
LIN {X 0,Y 467.128,Z 766.561,A -85,B 0,C 180,E1 -7640.911,E2 -7640.911} C_VEL
LIN {X 0,Y 466.883,Z 771.99,A -85,B 0,C 180,E1 -7642.214,E2 -7642.214} C_VEL
LIN {X 0,Y 466.835,Z 776.433,A -85,B 0,C 180,E1 -7643.517,E2 -7643.517} C_VEL
LIN {X 0,Y 466.732,Z 779.973,A -85,B 0,C 180,E1 -7644.817,E2 -7644.817} C_VEL
LIN {X 0,Y 466.636,Z 781.908,A -85,B 0,C 180,E1 -7645.681,E2 -7645.681} C_VEL
LIN {X 0,Y 466.659,Z 784.587,A -85,B 0,C 180,E1 -7647.411,E2 -7647.411} C_VEL
LIN {X 0,Y 466.616,Z 785.872,A -85,B 0,C 180,E1 -7649.137,E2 -7649.137} C_VEL
LIN {X 0,Y 466.597,Z 786.122,A -85,B 0,C 180,E1 -7650,E2 -7650} C_VEL
LIN {X 0,Y 466.604,Z 785.4,A -85,B 0,C 180,E1 -7651.726,E2 -7651.726} C_VEL
LIN {X 0,Y 466.659,Z 784.587,A -85,B 0,C 180,E1 -7652.589,E2 -7652.589} C_VEL
LIN {X 0,Y 466.636,Z 781.908,A -85,B 0,C 180,E1 -7654.319,E2 -7654.319} C_VEL
LIN {X 0,Y 466.757,Z 778.959,A -85,B 0,C 180,E1 -7655.616,E2 -7655.616} C_VEL
LIN {X 0,Y 466.824,Z 775.136,A -85,B 0,C 180,E1 -7656.917,E2 -7656.917} C_VEL
LIN {X 0,Y 466.966,Z 770.376,A -85,B 0,C 180,E1 -7658.22,E2 -7658.22} C_VEL
LIN {X 0,Y 467.258,Z 763.434,A -85,B 0,C 180,E1 -7659.742,E2 -7659.742} C_VEL
LIN {X 0,Y 467.613,Z 756.221,A -85,B 0,C 180,E1 -7661.047,E2 -7661.047} C_VEL
LIN {X 0,Y 467.97,Z 749.143,A -85,B 0,C 180,E1 -7662.137,E2 -7662.137} C_VEL
LIN {X 0,Y 468.34,Z 742.679,A -85,B 0,C 180,E1 -7663.008,E2 -7663.008} C_VEL
LIN {X 0,Y 468.867,Z 733.194,A -85,B 0,C 180,E1 -7664.097,E2 -7664.097} C_VEL
LIN {X 0,Y 469.38,Z 724.312,A -85,B 0,C 180,E1 -7664.968,E2 -7664.968} C_VEL
LIN {X 0,Y 469.966,Z 715.258,A -85,B 0,C 180,E1 -7665.726,E2 -7665.726} C_VEL
LIN {X 0,Y 470.564,Z 704.447,A -85,B 0,C 180,E1 -7666.485,E2 -7666.485} C_VEL
LIN {X 0,Y 471.101,Z 693.885,A -85,B 0,C 180,E1 -7667.095,E2 -7667.095} C_VEL
LIN {X 0,Y 471.491,Z 683.209,A -85,B 0,C 180,E1 -7667.596,E2 -7667.596} C_VEL
LIN {X 0,Y 471.879,Z 672.726,A -85,B 0,C 180,E1 -7667.979,E2 -7667.979} C_VEL
LIN {X 0,Y 472.229,Z 660.58,A -85,B 0,C 180,E1 -7668.296,E2 -7668.296} C_VEL
LIN {X 0,Y 472.641,Z 630.468,A -85,B 0,C 180,E1 -7668.785,E2 -7668.785} C_VEL
LIN {X 0,Y 473.28,Z 545.573,A -85,B 0,C 180,E1 -7670.095,E2 -7670.095} C_VEL
LIN {X 0,Y 468.974,Z 523.934,A -85,B 0,C 180,E1 -7670.66,E2 -7670.66} C_VEL
LIN {X 0,Y 469.735,Z 509.095,A -85,B 0,C 180,E1 -7673.592,E2 -7673.592} C_VEL
LIN {X 0,Y 470.321,Z 495.48,A -85,B 0,C 180,E1 -7676.288,E2 -7676.288} C_VEL
LIN {X 0,Y 468.491,Z 485.537,A -85,B 0,C 180,E1 -7678.457,E2 -7678.457} C_VEL
LIN {X 0,Y 467.605,Z 481.419,A -85,B 0,C 180,E1 -7679.437,E2 -7679.437} C_VEL
LIN {X 0,Y 467.582,Z 481.362,A -85,B 0,C 180,E1 -7682.758,E2 -7682.758} C_VEL
LIN {X 0,Y 467.551,Z 481.334,A -85,B 0,C 180,E1 -7685.889,E2 -7685.889} C_VEL
LIN {X 0,Y 467.58,Z 481.357,A -85,B 0,C 180,E1 -7689.144,E2 -7689.144} C_VEL
LIN {X 0,Y 467.583,Z 481.358,A -85,B 0,C 180,E1 -7692.566,E2 -7692.566} C_VEL
LIN {X 0,Y 467.567,Z 481.363,A -85,B 0,C 180,E1 -7695.052,E2 -7695.052} C_VEL
LIN {X 0,Y 467.585,Z 481.363,A -85,B 0,C 180,E1 -7697.439,E2 -7697.439} C_VEL
LIN {X 0,Y 467.608,Z 481.362,A -85,B 0,C 180,E1 -7700.858,E2 -7700.858} C_VEL
LIN {X 0,Y 467.558,Z 481.365,A -85,B 0,C 180,E1 -7704.26,E2 -7704.26} C_VEL
LIN {X 0,Y 467.576,Z 481.361,A -85,B 0,C 180,E1 -7707.32,E2 -7707.32} C_VEL
LIN {X 0,Y 467.564,Z 481.365,A -85,B 0,C 180,E1 -7710.667,E2 -7710.667} C_VEL
LIN {X 0,Y 467.621,Z 481.352,A -85,B 0,C 180,E1 -7713.2,E2 -7713.2} C_VEL
LIN {X 0,Y 467.585,Z 481.361,A -85,B 0,C 180,E1 -7716.467,E2 -7716.467} C_VEL
LIN {X 0,Y 467.616,Z 481.354,A -85,B 0,C 180,E1 -7719.777,E2 -7719.777} C_VEL
LIN {X 0,Y 467.601,Z 481.359,A -85,B 0,C 180,E1 -7722.506,E2 -7722.506} C_VEL
LIN {X 0,Y 467.598,Z 481.359,A -85,B 0,C 180,E1 -7725.196,E2 -7725.196} C_VEL
LIN {X 0,Y 467.647,Z 481.353,A -85,B 0,C 180,E1 -7727.854,E2 -7727.854} C_VEL
LIN {X 0,Y 467.673,Z 481.357,A -85,B 0,C 180,E1 -7731.357,E2 -7731.357} C_VEL
LIN {X 0,Y 467.735,Z 481.33,A -85,B 0,C 180,E1 -7733.962,E2 -7733.962} C_VEL
LIN {X 0,Y 467.851,Z 481.332,A -85,B 0,C 180,E1 -7737.417,E2 -7737.417} C_VEL
LIN {X 0,Y 467.873,Z 481.321,A -85,B 0,C 180,E1 -7740,E2 -7740} C_VEL
LIN {X 0,Y 467.851,Z 481.315,A -85,B 0,C 180,E1 -7742.583,E2 -7742.583} C_VEL
LIN {X 0,Y 467.734,Z 481.344,A -85,B 0,C 180,E1 -7746.037,E2 -7746.037} C_VEL
LIN {X 0,Y 467.673,Z 481.343,A -85,B 0,C 180,E1 -7748.642,E2 -7748.642} C_VEL
LIN {X 0,Y 467.647,Z 481.354,A -85,B 0,C 180,E1 -7752.145,E2 -7752.145} C_VEL
LIN {X 0,Y 467.629,Z 481.355,A -85,B 0,C 180,E1 -7755.695,E2 -7755.695} C_VEL
LIN {X 0,Y 467.608,Z 481.353,A -85,B 0,C 180,E1 -7758.765,E2 -7758.765} C_VEL
LIN {X 0,Y 467.57,Z 481.367,A -85,B 0,C 180,E1 -7761.268,E2 -7761.268} C_VEL
LIN {X 0,Y 467.563,Z 481.357,A -85,B 0,C 180,E1 -7763.943,E2 -7763.943} C_VEL
LIN {X 0,Y 467.618,Z 481.357,A -85,B 0,C 180,E1 -7766.8,E2 -7766.8} C_VEL
LIN {X 0,Y 467.578,Z 481.36,A -85,B 0,C 180,E1 -7769.736,E2 -7769.736} C_VEL
LIN {X 0,Y 467.575,Z 481.363,A -85,B 0,C 180,E1 -7772.758,E2 -7772.758} C_VEL
LIN {X 0,Y 467.548,Z 481.365,A -85,B 0,C 180,E1 -7775.889,E2 -7775.889} C_VEL
LIN {X 0,Y 467.574,Z 481.365,A -85,B 0,C 180,E1 -7779.145,E2 -7779.145} C_VEL
LIN {X 0,Y 467.611,Z 481.359,A -85,B 0,C 180,E1 -7782.572,E2 -7782.572} C_VEL
LIN {X 0,Y 467.566,Z 481.344,A -85,B 0,C 180,E1 -7786.177,E2 -7786.177} C_VEL
LIN {X 0,Y 467.584,Z 481.358,A -85,B 0,C 180,E1 -7788.722,E2 -7788.722} C_VEL
LIN {X 0,Y 467.572,Z 481.367,A -85,B 0,C 180,E1 -7791.407,E2 -7791.407} C_VEL
LIN {X 0,Y 467.556,Z 481.362,A -85,B 0,C 180,E1 -7794.261,E2 -7794.261} C_VEL
LIN {X 0,Y 467.576,Z 481.367,A -85,B 0,C 180,E1 -7797.321,E2 -7797.321} C_VEL
LIN {X 0,Y 467.572,Z 481.365,A -85,B 0,C 180,E1 -7800.666,E2 -7800.666} C_VEL
LIN {X 0,Y 467.611,Z 481.362,A -85,B 0,C 180,E1 -7803.2,E2 -7803.2} C_VEL
LIN {X 0,Y 467.588,Z 481.365,A -85,B 0,C 180,E1 -7806.468,E2 -7806.468} C_VEL
LIN {X 0,Y 467.618,Z 481.364,A -85,B 0,C 180,E1 -7809.777,E2 -7809.777} C_VEL
LIN {X 0,Y 467.604,Z 481.364,A -85,B 0,C 180,E1 -7812.507,E2 -7812.507} C_VEL
LIN {X 0,Y 467.592,Z 481.364,A -85,B 0,C 180,E1 -7815.434,E2 -7815.434} C_VEL
LIN {X 0,Y 466.923,Z 481.451,A -85,B 0,C 180,E1 -7816.153,E2 -7816.153} C_VEL
LIN {X 0,Y 464.079,Z 481.803,A -85,B 0,C 180,E1 -7817.321,E2 -7817.321} C_VEL
LIN {X 0,Y 461.68,Z 482.104,A -85,B 0,C 180,E1 -7818.264,E2 -7818.264} C_VEL
LIN {X 0,Y 460.654,Z 482.228,A -85,B 0,C 180,E1 -7818.991,E2 -7818.991} C_VEL
LIN {X 0,Y 460.573,Z 482.239,A -85,B 0,C 180,E1 -7819.238,E2 -7819.238} C_VEL
LIN {X 0,Y 460.716,Z 482.222,A -85,B 0,C 180,E1 -7822.538,E2 -7822.538} C_VEL
LIN {X 0,Y 460.693,Z 482.224,A -85,B 0,C 180,E1 -7824.748,E2 -7824.748} C_VEL
LIN {X 0,Y 460.822,Z 482.21,A -85,B 0,C 180,E1 -7827.378,E2 -7827.378} C_VEL
LIN {X 0,Y 460.85,Z 482.208,A -85,B 0,C 180,E1 -7830,E2 -7830} C_VEL
LIN {X 0,Y 460.821,Z 482.21,A -85,B 0,C 180,E1 -7832.622,E2 -7832.622} C_VEL
LIN {X 0,Y 460.706,Z 482.225,A -85,B 0,C 180,E1 -7836.13,E2 -7836.13} C_VEL
LIN {X 0,Y 460.625,Z 482.232,A -85,B 0,C 180,E1 -7838.776,E2 -7838.776} C_VEL
LIN {X 0,Y 460.609,Z 482.236,A -85,B 0,C 180,E1 -7842.445,E2 -7842.445} C_VEL
LIN {X 0,Y 460.596,Z 482.239,A -85,B 0,C 180,E1 -7845.997,E2 -7845.997} C_VEL
LIN {X 0,Y 460.566,Z 482.239,A -85,B 0,C 180,E1 -7848.902,E2 -7848.902} C_VEL
LIN {X 0,Y 460.511,Z 482.246,A -85,B 0,C 180,E1 -7851.485,E2 -7851.485} C_VEL
LIN {X 0,Y 460.538,Z 482.246,A -85,B 0,C 180,E1 -7854.332,E2 -7854.332} C_VEL
LIN {X 0,Y 460.574,Z 482.238,A -85,B 0,C 180,E1 -7857.243,E2 -7857.243} C_VEL
LIN {X 0,Y 460.521,Z 482.249,A -85,B 0,C 180,E1 -7860.238,E2 -7860.238} C_VEL
LIN {X 0,Y 460.523,Z 482.243,A -85,B 0,C 180,E1 -7863.324,E2 -7863.324} C_VEL
LIN {X 0,Y 460.472,Z 482.236,A -85,B 0,C 180,E1 -7866.529,E2 -7866.529} C_VEL
LIN {X 0,Y 460.571,Z 482.24,A -85,B 0,C 180,E1 -7869.857,E2 -7869.857} C_VEL
LIN {X 0,Y 460.534,Z 482.215,A -85,B 0,C 180,E1 -7872.904,E2 -7872.904} C_VEL
LIN {X 0,Y 460.516,Z 482.241,A -85,B 0,C 180,E1 -7875.828,E2 -7875.828} C_VEL
LIN {X 0,Y 460.526,Z 482.235,A -85,B 0,C 180,E1 -7878.989,E2 -7878.989} C_VEL
LIN {X 0,Y 460.518,Z 482.243,A -85,B 0,C 180,E1 -7881.267,E2 -7881.267} C_VEL
LIN {X 0,Y 460.505,Z 482.244,A -85,B 0,C 180,E1 -7884.555,E2 -7884.555} C_VEL
LIN {X 0,Y 460.523,Z 482.242,A -85,B 0,C 180,E1 -7887.716,E2 -7887.716} C_VEL
LIN {X 0,Y 460.538,Z 482.241,A -85,B 0,C 180,E1 -7890.77,E2 -7890.77} C_VEL
LIN {X 0,Y 460.558,Z 482.237,A -85,B 0,C 180,E1 -7893.735,E2 -7893.735} C_VEL
LIN {X 0,Y 460.536,Z 482.238,A -85,B 0,C 180,E1 -7896.624,E2 -7896.624} C_VEL
LIN {X 0,Y 460.542,Z 482.239,A -85,B 0,C 180,E1 -7899.453,E2 -7899.453} C_VEL
LIN {X 0,Y 460.549,Z 482.232,A -85,B 0,C 180,E1 -7902.23,E2 -7902.23} C_VEL
LIN {X 0,Y 460.555,Z 482.238,A -85,B 0,C 180,E1 -7904.965,E2 -7904.965} C_VEL
LIN {X 0,Y 460.603,Z 482.227,A -85,B 0,C 180,E1 -7908.56,E2 -7908.56} C_VEL
LIN {X 0,Y 460.685,Z 482.217,A -85,B 0,C 180,E1 -7912.109,E2 -7912.109} C_VEL
LIN {X 0,Y 460.696,Z 482.221,A -85,B 0,C 180,E1 -7914.749,E2 -7914.749} C_VEL
LIN {X 0,Y 460.816,Z 482.19,A -85,B 0,C 180,E1 -7917.378,E2 -7917.378} C_VEL
LIN {X 0,Y 460.843,Z 482.196,A -85,B 0,C 180,E1 -7920,E2 -7920} C_VEL
LIN {X 0,Y 460.817,Z 482.207,A -85,B 0,C 180,E1 -7922.623,E2 -7922.623} C_VEL
LIN {X 0,Y 460.701,Z 482.206,A -85,B 0,C 180,E1 -7926.13,E2 -7926.13} C_VEL
LIN {X 0,Y 460.62,Z 482.234,A -85,B 0,C 180,E1 -7928.777,E2 -7928.777} C_VEL
LIN {X 0,Y 460.605,Z 482.226,A -85,B 0,C 180,E1 -7932.446,E2 -7932.446} C_VEL
LIN {X 0,Y 460.592,Z 482.231,A -85,B 0,C 180,E1 -7935.998,E2 -7935.998} C_VEL
LIN {X 0,Y 460.563,Z 482.234,A -85,B 0,C 180,E1 -7938.902,E2 -7938.902} C_VEL
LIN {X 0,Y 460.508,Z 482.236,A -85,B 0,C 180,E1 -7941.486,E2 -7941.486} C_VEL
LIN {X 0,Y 460.535,Z 482.244,A -85,B 0,C 180,E1 -7944.333,E2 -7944.333} C_VEL
LIN {X 0,Y 460.577,Z 482.227,A -85,B 0,C 180,E1 -7947.244,E2 -7947.244} C_VEL
LIN {X 0,Y 460.505,Z 482.246,A -85,B 0,C 180,E1 -7950.241,E2 -7950.241} C_VEL
LIN {X 0,Y 460.524,Z 482.237,A -85,B 0,C 180,E1 -7953.326,E2 -7953.326} C_VEL
LIN {X 0,Y 460.474,Z 482.254,A -85,B 0,C 180,E1 -7956.53,E2 -7956.53} C_VEL
LIN {X 0,Y 460.569,Z 482.237,A -85,B 0,C 180,E1 -7959.859,E2 -7959.859} C_VEL
LIN {X 0,Y 460.509,Z 482.25,A -85,B 0,C 180,E1 -7962.901,E2 -7962.901} C_VEL
LIN {X 0,Y 460.516,Z 482.236,A -85,B 0,C 180,E1 -7965.83,E2 -7965.83} C_VEL
LIN {X 0,Y 460.531,Z 482.247,A -85,B 0,C 180,E1 -7968.99,E2 -7968.99} C_VEL
LIN {X 0,Y 460.524,Z 482.23,A -85,B 0,C 180,E1 -7971.268,E2 -7971.268} C_VEL
LIN {X 0,Y 460.508,Z 482.217,A -85,B 0,C 180,E1 -7974.555,E2 -7974.555} C_VEL
LIN {X 0,Y 460.531,Z 482.234,A -85,B 0,C 180,E1 -7977.716,E2 -7977.716} C_VEL
LIN {X 0,Y 460.592,Z 482.372,A -85,B 0,C 180,E1 -7980.335,E2 -7980.335} C_VEL
LIN {X 0,Y 462.85,Z 493.547,A -85,B 0,C 180,E1 -7982.902,E2 -7982.902} C_VEL
LIN {X 0,Y 463.407,Z 498.245,A -85,B 0,C 180,E1 -7983.909,E2 -7983.909} C_VEL
LIN {X 0,Y 462.645,Z 512.246,A -85,B 0,C 180,E1 -7986.737,E2 -7986.737} C_VEL
LIN {X 0,Y 462.047,Z 523.559,A -85,B 0,C 180,E1 -7988.998,E2 -7988.998} C_VEL
LIN {X 0,Y 462.98,Z 528.314,A -85,B 0,C 180,E1 -7989.163,E2 -7989.163} C_VEL
LIN {X 0,Y 466.694,Z 547.116,A -85,B 0,C 180,E1 -7989.637,E2 -7989.637} C_VEL
LIN {X 0,Y 465.597,Z 656.304,A -85,B 0,C 180,E1 -7991.349,E2 -7991.349} C_VEL
LIN {X 0,Y 465.281,Z 668.15,A -85,B 0,C 180,E1 -7991.621,E2 -7991.621} C_VEL
LIN {X 0,Y 464.832,Z 679.605,A -85,B 0,C 180,E1 -7992.001,E2 -7992.001} C_VEL
LIN {X 0,Y 464.436,Z 690.807,A -85,B 0,C 180,E1 -7992.5,E2 -7992.5} C_VEL
LIN {X 0,Y 463.877,Z 701.42,A -85,B 0,C 180,E1 -7993.088,E2 -7993.088} C_VEL
LIN {X 0,Y 463.36,Z 710.663,A -85,B 0,C 180,E1 -7993.705,E2 -7993.705} C_VEL
LIN {X 0,Y 462.72,Z 720.39,A -85,B 0,C 180,E1 -7994.473,E2 -7994.473} C_VEL
LIN {X 0,Y 462.157,Z 729.815,A -85,B 0,C 180,E1 -7995.356,E2 -7995.356} C_VEL
LIN {X 0,Y 461.589,Z 738.84,A -85,B 0,C 180,E1 -7996.35,E2 -7996.35} C_VEL
LIN {X 0,Y 461.139,Z 746.034,A -85,B 0,C 180,E1 -7997.264,E2 -7997.264} C_VEL
LIN {X 0,Y 460.794,Z 753.347,A -85,B 0,C 180,E1 -7998.341,E2 -7998.341} C_VEL
LIN {X 0,Y 460.31,Z 760.958,A -85,B 0,C 180,E1 -7999.666,E2 -7999.666} C_VEL
LIN {X 0,Y 460.071,Z 766.361,A -85,B 0,C 180,E1 -8000.77,E2 -8000.77} C_VEL
LIN {X 0,Y 459.822,Z 771.792,A -85,B 0,C 180,E1 -8002.094,E2 -8002.094} C_VEL
LIN {X 0,Y 459.735,Z 774.937,A -85,B 0,C 180,E1 -8002.976,E2 -8002.976} C_VEL
LIN {X 0,Y 459.646,Z 779.775,A -85,B 0,C 180,E1 -8004.736,E2 -8004.736} C_VEL
LIN {X 0,Y 459.553,Z 781.71,A -85,B 0,C 180,E1 -8005.615,E2 -8005.615} C_VEL
LIN {X 0,Y 459.581,Z 784.389,A -85,B 0,C 180,E1 -8007.371,E2 -8007.371} C_VEL
LIN {X 0,Y 459.519,Z 785.674,A -85,B 0,C 180,E1 -8009.124,E2 -8009.124} C_VEL
LIN {X 0,Y 459.529,Z 785.925,A -85,B 0,C 180,E1 -8010,E2 -8010} C_VEL
LIN {X 0,Y 459.517,Z 785.202,A -85,B 0,C 180,E1 -8011.753,E2 -8011.753} C_VEL
LIN {X 0,Y 459.581,Z 784.389,A -85,B 0,C 180,E1 -8012.629,E2 -8012.629} C_VEL
LIN {X 0,Y 459.553,Z 781.71,A -85,B 0,C 180,E1 -8014.385,E2 -8014.385} C_VEL
LIN {X 0,Y 459.655,Z 778.76,A -85,B 0,C 180,E1 -8015.704,E2 -8015.704} C_VEL
LIN {X 0,Y 459.734,Z 774.937,A -85,B 0,C 180,E1 -8017.025,E2 -8017.025} C_VEL
LIN {X 0,Y 459.912,Z 770.177,A -85,B 0,C 180,E1 -8018.347,E2 -8018.347} C_VEL
LIN {X 0,Y 460.214,Z 763.234,A -85,B 0,C 180,E1 -8019.892,E2 -8019.892} C_VEL
LIN {X 0,Y 460.607,Z 756.022,A -85,B 0,C 180,E1 -8021.218,E2 -8021.218} C_VEL
LIN {X 0,Y 460.992,Z 748.944,A -85,B 0,C 180,E1 -8022.323,E2 -8022.323} C_VEL
LIN {X 0,Y 461.443,Z 740.659,A -85,B 0,C 180,E1 -8023.43,E2 -8023.43} C_VEL
LIN {X 0,Y 462.02,Z 731.935,A -85,B 0,C 180,E1 -8024.423,E2 -8024.423} C_VEL
LIN {X 0,Y 462.559,Z 722.872,A -85,B 0,C 180,E1 -8025.307,E2 -8025.307} C_VEL
LIN {X 0,Y 463.188,Z 713.594,A -85,B 0,C 180,E1 -8026.075,E2 -8026.075} C_VEL
LIN {X 0,Y 463.735,Z 704.248,A -85,B 0,C 180,E1 -8026.735,E2 -8026.735} C_VEL
LIN {X 0,Y 464.291,Z 693.623,A -85,B 0,C 180,E1 -8027.357,E2 -8027.357} C_VEL
LIN {X 0,Y 464.732,Z 682.327,A -85,B 0,C 180,E1 -8027.889,E2 -8027.889} C_VEL
LIN {X 0,Y 465.157,Z 671.798,A -85,B 0,C 180,E1 -8028.27,E2 -8028.27} C_VEL
LIN {X 0,Y 465.491,Z 660.382,A -85,B 0,C 180,E1 -8028.57,E2 -8028.57} C_VEL
LIN {X 0,Y 465.937,Z 630.271,A -85,B 0,C 180,E1 -8029.065,E2 -8029.065} C_VEL
LIN {X 0,Y 466.606,Z 546.6,A -85,B 0,C 180,E1 -8030.376,E2 -8030.376} C_VEL
LIN {X 0,Y 462.043,Z 523.92,A -85,B 0,C 180,E1 -8030.97,E2 -8030.97} C_VEL
LIN {X 0,Y 462.065,Z 522.558,A -85,B 0,C 180,E1 -8031.176,E2 -8031.176} C_VEL
LIN {X 0,Y 462.871,Z 508.925,A -85,B 0,C 180,E1 -8033.963,E2 -8033.963} C_VEL
LIN {X 0,Y 463.427,Z 498.333,A -85,B 0,C 180,E1 -8036.09,E2 -8036.09} C_VEL
LIN {X 0,Y 462.896,Z 493.593,A -85,B 0,C 180,E1 -8037.095,E2 -8037.095} C_VEL
LIN {X 0,Y 460.592,Z 482.375,A -85,B 0,C 180,E1 -8039.665,E2 -8039.665} C_VEL
LIN {X 0,Y 460.53,Z 482.242,A -85,B 0,C 180,E1 -8042.929,E2 -8042.929} C_VEL
LIN {X 0,Y 460.495,Z 482.21,A -85,B 0,C 180,E1 -8046.013,E2 -8046.013} C_VEL
LIN {X 0,Y 460.542,Z 482.229,A -85,B 0,C 180,E1 -8048.897,E2 -8048.897} C_VEL
LIN {X 0,Y 460.521,Z 482.237,A -85,B 0,C 180,E1 -8052.18,E2 -8052.18} C_VEL
LIN {X 0,Y 460.512,Z 482.247,A -85,B 0,C 180,E1 -8055.411,E2 -8055.411} C_VEL
LIN {X 0,Y 460.531,Z 482.237,A -85,B 0,C 180,E1 -8058.396,E2 -8058.396} C_VEL
LIN {X 0,Y 460.537,Z 482.241,A -85,B 0,C 180,E1 -8061.268,E2 -8061.268} C_VEL
LIN {X 0,Y 460.508,Z 482.244,A -85,B 0,C 180,E1 -8064.554,E2 -8064.554} C_VEL
LIN {X 0,Y 460.526,Z 482.242,A -85,B 0,C 180,E1 -8067.715,E2 -8067.715} C_VEL
LIN {X 0,Y 460.534,Z 482.241,A -85,B 0,C 180,E1 -8070.768,E2 -8070.768} C_VEL
LIN {X 0,Y 460.562,Z 482.237,A -85,B 0,C 180,E1 -8073.734,E2 -8073.734} C_VEL
LIN {X 0,Y 460.539,Z 482.24,A -85,B 0,C 180,E1 -8076.623,E2 -8076.623} C_VEL
LIN {X 0,Y 460.544,Z 482.232,A -85,B 0,C 180,E1 -8079.452,E2 -8079.452} C_VEL
LIN {X 0,Y 460.551,Z 482.238,A -85,B 0,C 180,E1 -8082.229,E2 -8082.229} C_VEL
LIN {X 0,Y 460.557,Z 482.237,A -85,B 0,C 180,E1 -8084.964,E2 -8084.964} C_VEL
LIN {X 0,Y 460.602,Z 482.228,A -85,B 0,C 180,E1 -8088.559,E2 -8088.559} C_VEL
LIN {X 0,Y 460.686,Z 482.217,A -85,B 0,C 180,E1 -8092.108,E2 -8092.108} C_VEL
LIN {X 0,Y 460.689,Z 482.206,A -85,B 0,C 180,E1 -8094.748,E2 -8094.748} C_VEL
LIN {X 0,Y 460.816,Z 482.207,A -85,B 0,C 180,E1 -8097.377,E2 -8097.377} C_VEL
LIN {X 0,Y 460.843,Z 482.196,A -85,B 0,C 180,E1 -8100,E2 -8100} C_VEL
LIN {X 0,Y 460.816,Z 482.191,A -85,B 0,C 180,E1 -8102.622,E2 -8102.622} C_VEL
LIN {X 0,Y 460.7,Z 482.219,A -85,B 0,C 180,E1 -8106.13,E2 -8106.13} C_VEL
LIN {X 0,Y 460.62,Z 482.222,A -85,B 0,C 180,E1 -8108.776,E2 -8108.776} C_VEL
LIN {X 0,Y 460.603,Z 482.23,A -85,B 0,C 180,E1 -8112.445,E2 -8112.445} C_VEL
LIN {X 0,Y 460.59,Z 482.227,A -85,B 0,C 180,E1 -8115.997,E2 -8115.997} C_VEL
LIN {X 0,Y 460.561,Z 482.231,A -85,B 0,C 180,E1 -8118.902,E2 -8118.902} C_VEL
LIN {X 0,Y 460.506,Z 482.25,A -85,B 0,C 180,E1 -8121.486,E2 -8121.486} C_VEL
LIN {X 0,Y 460.532,Z 482.231,A -85,B 0,C 180,E1 -8124.332,E2 -8124.332} C_VEL
LIN {X 0,Y 460.574,Z 482.237,A -85,B 0,C 180,E1 -8127.243,E2 -8127.243} C_VEL
LIN {X 0,Y 460.518,Z 482.234,A -85,B 0,C 180,E1 -8130.239,E2 -8130.239} C_VEL
LIN {X 0,Y 460.52,Z 482.245,A -85,B 0,C 180,E1 -8133.325,E2 -8133.325} C_VEL
LIN {X 0,Y 460.47,Z 482.244,A -85,B 0,C 180,E1 -8136.529,E2 -8136.529} C_VEL
LIN {X 0,Y 460.55,Z 482.238,A -85,B 0,C 180,E1 -8139.86,E2 -8139.86} C_VEL
LIN {X 0,Y 460.534,Z 482.241,A -85,B 0,C 180,E1 -8142.905,E2 -8142.905} C_VEL
LIN {X 0,Y 460.516,Z 482.226,A -85,B 0,C 180,E1 -8145.829,E2 -8145.829} C_VEL
LIN {X 0,Y 460.538,Z 482.236,A -85,B 0,C 180,E1 -8148.991,E2 -8148.991} C_VEL
LIN {X 0,Y 460.542,Z 482.242,A -85,B 0,C 180,E1 -8151.27,E2 -8151.27} C_VEL
LIN {X 0,Y 460.507,Z 482.242,A -85,B 0,C 180,E1 -8154.555,E2 -8154.555} C_VEL
LIN {X 0,Y 460.526,Z 482.248,A -85,B 0,C 180,E1 -8157.716,E2 -8157.716} C_VEL
LIN {X 0,Y 460.541,Z 482.241,A -85,B 0,C 180,E1 -8160.77,E2 -8160.77} C_VEL
LIN {X 0,Y 460.558,Z 482.244,A -85,B 0,C 180,E1 -8163.735,E2 -8163.735} C_VEL
LIN {X 0,Y 460.541,Z 482.242,A -85,B 0,C 180,E1 -8166.624,E2 -8166.624} C_VEL
LIN {X 0,Y 460.547,Z 482.244,A -85,B 0,C 180,E1 -8169.453,E2 -8169.453} C_VEL
LIN {X 0,Y 460.555,Z 482.243,A -85,B 0,C 180,E1 -8172.23,E2 -8172.23} C_VEL
LIN {X 0,Y 460.561,Z 482.24,A -85,B 0,C 180,E1 -8174.965,E2 -8174.965} C_VEL
LIN {X 0,Y 460.607,Z 482.235,A -85,B 0,C 180,E1 -8178.559,E2 -8178.559} C_VEL
LIN {X 0,Y 460.573,Z 482.239,A -85,B 0,C 180,E1 -8179.238,E2 -8179.238} C_VEL
LIN {X 0,Y 459.919,Z 482.324,A -85,B 0,C 180,E1 -8179.968,E2 -8179.968} C_VEL
LIN {X 0,Y 457.101,Z 482.674,A -85,B 0,C 180,E1 -8181.154,E2 -8181.154} C_VEL
LIN {X 0,Y 454.722,Z 482.971,A -85,B 0,C 180,E1 -8182.112,E2 -8182.112} C_VEL
LIN {X 0,Y 453.71,Z 483.094,A -85,B 0,C 180,E1 -8182.85,E2 -8182.85} C_VEL
LIN {X 0,Y 453.633,Z 483.102,A -85,B 0,C 180,E1 -8183.101,E2 -8183.101} C_VEL
LIN {X 0,Y 453.667,Z 483.1,A -85,B 0,C 180,E1 -8184.667,E2 -8184.667} C_VEL
LIN {X 0,Y 453.762,Z 483.089,A -85,B 0,C 180,E1 -8187.337,E2 -8187.337} C_VEL
LIN {X 0,Y 453.82,Z 483.084,A -85,B 0,C 180,E1 -8190,E2 -8190} C_VEL
LIN {X 0,Y 453.762,Z 483.089,A -85,B 0,C 180,E1 -8192.663,E2 -8192.663} C_VEL
LIN {X 0,Y 453.673,Z 483.101,A -85,B 0,C 180,E1 -8196.225,E2 -8196.225} C_VEL
LIN {X 0,Y 453.588,Z 483.108,A -85,B 0,C 180,E1 -8198.913,E2 -8198.913} C_VEL
LIN {X 0,Y 453.559,Z 483.114,A -85,B 0,C 180,E1 -8202.529,E2 -8202.529} C_VEL
LIN {X 0,Y 453.54,Z 483.118,A -85,B 0,C 180,E1 -8206.196,E2 -8206.196} C_VEL
LIN {X 0,Y 453.515,Z 483.118,A -85,B 0,C 180,E1 -8209.04,E2 -8209.04} C_VEL
LIN {X 0,Y 453.472,Z 483.126,A -85,B 0,C 180,E1 -8211.836,E2 -8211.836} C_VEL
LIN {X 0,Y 453.509,Z 483.119,A -85,B 0,C 180,E1 -8214.734,E2 -8214.734} C_VEL
LIN {X 0,Y 453.533,Z 483.119,A -85,B 0,C 180,E1 -8217.961,E2 -8217.961} C_VEL
LIN {X 0,Y 453.477,Z 483.122,A -85,B 0,C 180,E1 -8220.759,E2 -8220.759} C_VEL
LIN {X 0,Y 453.472,Z 483.126,A -85,B 0,C 180,E1 -8223.912,E2 -8223.912} C_VEL
LIN {X 0,Y 453.465,Z 483.109,A -85,B 0,C 180,E1 -8227.187,E2 -8227.187} C_VEL
LIN {X 0,Y 453.526,Z 483.114,A -85,B 0,C 180,E1 -8229.445,E2 -8229.445} C_VEL
LIN {X 0,Y 453.484,Z 483.092,A -85,B 0,C 180,E1 -8232.991,E2 -8232.991} C_VEL
LIN {X 0,Y 453.469,Z 483.118,A -85,B 0,C 180,E1 -8235.78,E2 -8235.78} C_VEL
LIN {X 0,Y 453.485,Z 483.12,A -85,B 0,C 180,E1 -8238.211,E2 -8238.211} C_VEL
LIN {X 0,Y 453.507,Z 483.118,A -85,B 0,C 180,E1 -8240.79,E2 -8240.79} C_VEL
LIN {X 0,Y 453.448,Z 483.12,A -85,B 0,C 180,E1 -8243.917,E2 -8243.917} C_VEL
LIN {X 0,Y 453.474,Z 483.119,A -85,B 0,C 180,E1 -8247.151,E2 -8247.151} C_VEL
LIN {X 0,Y 453.505,Z 483.112,A -85,B 0,C 180,E1 -8250.271,E2 -8250.271} C_VEL
LIN {X 0,Y 453.504,Z 483.115,A -85,B 0,C 180,E1 -8253.294,E2 -8253.294} C_VEL
LIN {X 0,Y 453.493,Z 483.11,A -85,B 0,C 180,E1 -8256.239,E2 -8256.239} C_VEL
LIN {X 0,Y 453.473,Z 483.12,A -85,B 0,C 180,E1 -8259.118,E2 -8259.118} C_VEL
LIN {X 0,Y 453.502,Z 483.111,A -85,B 0,C 180,E1 -8261.945,E2 -8261.945} C_VEL
LIN {X 0,Y 453.529,Z 483.116,A -85,B 0,C 180,E1 -8264.726,E2 -8264.726} C_VEL
LIN {X 0,Y 453.551,Z 483.108,A -85,B 0,C 180,E1 -8268.379,E2 -8268.379} C_VEL
LIN {X 0,Y 453.642,Z 483.093,A -85,B 0,C 180,E1 -8271.986,E2 -8271.986} C_VEL
LIN {X 0,Y 453.669,Z 483.097,A -85,B 0,C 180,E1 -8274.667,E2 -8274.667} C_VEL
LIN {X 0,Y 453.757,Z 483.069,A -85,B 0,C 180,E1 -8277.337,E2 -8277.337} C_VEL
LIN {X 0,Y 453.814,Z 483.072,A -85,B 0,C 180,E1 -8280,E2 -8280} C_VEL
LIN {X 0,Y 453.757,Z 483.086,A -85,B 0,C 180,E1 -8282.664,E2 -8282.664} C_VEL
LIN {X 0,Y 453.669,Z 483.082,A -85,B 0,C 180,E1 -8286.226,E2 -8286.226} C_VEL
LIN {X 0,Y 453.584,Z 483.109,A -85,B 0,C 180,E1 -8288.914,E2 -8288.914} C_VEL
LIN {X 0,Y 453.555,Z 483.102,A -85,B 0,C 180,E1 -8292.529,E2 -8292.529} C_VEL
LIN {X 0,Y 453.537,Z 483.112,A -85,B 0,C 180,E1 -8296.197,E2 -8296.197} C_VEL
LIN {X 0,Y 453.512,Z 483.11,A -85,B 0,C 180,E1 -8299.041,E2 -8299.041} C_VEL
LIN {X 0,Y 453.469,Z 483.113,A -85,B 0,C 180,E1 -8301.837,E2 -8301.837} C_VEL
LIN {X 0,Y 453.507,Z 483.119,A -85,B 0,C 180,E1 -8304.735,E2 -8304.735} C_VEL
LIN {X 0,Y 453.531,Z 483.104,A -85,B 0,C 180,E1 -8307.962,E2 -8307.962} C_VEL
LIN {X 0,Y 453.46,Z 483.119,A -85,B 0,C 180,E1 -8311.526,E2 -8311.526} C_VEL
LIN {X 0,Y 453.484,Z 483.123,A -85,B 0,C 180,E1 -8314.778,E2 -8314.778} C_VEL
LIN {X 0,Y 453.477,Z 483.116,A -85,B 0,C 180,E1 -8318.311,E2 -8318.311} C_VEL
LIN {X 0,Y 453.512,Z 483.122,A -85,B 0,C 180,E1 -8320.607,E2 -8320.607} C_VEL
LIN {X 0,Y 453.46,Z 483.125,A -85,B 0,C 180,E1 -8324.222,E2 -8324.222} C_VEL
LIN {X 0,Y 453.464,Z 483.111,A -85,B 0,C 180,E1 -8327.006,E2 -8327.006} C_VEL
LIN {X 0,Y 453.515,Z 483.113,A -85,B 0,C 180,E1 -8330.554,E2 -8330.554} C_VEL
LIN {X 0,Y 453.452,Z 483.085,A -85,B 0,C 180,E1 -8333.918,E2 -8333.918} C_VEL
LIN {X 0,Y 453.482,Z 483.119,A -85,B 0,C 180,E1 -8337.152,E2 -8337.152} C_VEL
LIN {X 0,Y 453.533,Z 483.235,A -85,B 0,C 180,E1 -8340.043,E2 -8340.043} C_VEL
LIN {X 0,Y 455.613,Z 493.351,A -85,B 0,C 180,E1 -8342.435,E2 -8342.435} C_VEL
LIN {X 0,Y 456.443,Z 498.047,A -85,B 0,C 180,E1 -8343.48,E2 -8343.48} C_VEL
LIN {X 0,Y 455.862,Z 510.89,A -85,B 0,C 180,E1 -8346.129,E2 -8346.129} C_VEL
LIN {X 0,Y 455.115,Z 523.497,A -85,B 0,C 180,E1 -8348.679,E2 -8348.679} C_VEL
LIN {X 0,Y 458.514,Z 540.334,A -85,B 0,C 180,E1 -8349.15,E2 -8349.15} C_VEL
LIN {X 0,Y 460.005,Z 548.008,A -85,B 0,C 180,E1 -8349.345,E2 -8349.345} C_VEL
LIN {X 0,Y 458.845,Z 657.465,A -85,B 0,C 180,E1 -8351.093,E2 -8351.093} C_VEL
LIN {X 0,Y 458.521,Z 668.864,A -85,B 0,C 180,E1 -8351.369,E2 -8351.369} C_VEL
LIN {X 0,Y 458.069,Z 679.407,A -85,B 0,C 180,E1 -8351.726,E2 -8351.726} C_VEL
LIN {X 0,Y 457.659,Z 689.913,A -85,B 0,C 180,E1 -8352.195,E2 -8352.195} C_VEL
LIN {X 0,Y 457.102,Z 700.128,A -85,B 0,C 180,E1 -8352.758,E2 -8352.758} C_VEL
LIN {X 0,Y 456.509,Z 710.464,A -85,B 0,C 180,E1 -8353.453,E2 -8353.453} C_VEL
LIN {X 0,Y 455.867,Z 720.192,A -85,B 0,C 180,E1 -8354.234,E2 -8354.234} C_VEL
LIN {X 0,Y 455.211,Z 729.615,A -85,B 0,C 180,E1 -8355.128,E2 -8355.128} C_VEL
LIN {X 0,Y 454.63,Z 738.641,A -85,B 0,C 180,E1 -8356.137,E2 -8356.137} C_VEL
LIN {X 0,Y 454.125,Z 746.477,A -85,B 0,C 180,E1 -8357.158,E2 -8357.158} C_VEL
LIN {X 0,Y 453.702,Z 754.485,A -85,B 0,C 180,E1 -8358.383,E2 -8358.383} C_VEL
LIN {X 0,Y 453.26,Z 760.758,A -85,B 0,C 180,E1 -8359.503,E2 -8359.503} C_VEL
LIN {X 0,Y 453.007,Z 766.162,A -85,B 0,C 180,E1 -8360.625,E2 -8360.625} C_VEL
LIN {X 0,Y 452.752,Z 771.592,A -85,B 0,C 180,E1 -8361.969,E2 -8361.969} C_VEL
LIN {X 0,Y 452.658,Z 774.738,A -85,B 0,C 180,E1 -8362.865,E2 -8362.865} C_VEL
LIN {X 0,Y 452.561,Z 779.576,A -85,B 0,C 180,E1 -8364.654,E2 -8364.654} C_VEL
LIN {X 0,Y 452.473,Z 781.512,A -85,B 0,C 180,E1 -8365.546,E2 -8365.546} C_VEL
LIN {X 0,Y 452.504,Z 784.192,A -85,B 0,C 180,E1 -8367.329,E2 -8367.329} C_VEL
LIN {X 0,Y 452.426,Z 785.476,A -85,B 0,C 180,E1 -8369.11,E2 -8369.11} C_VEL
LIN {X 0,Y 452.433,Z 785.727,A -85,B 0,C 180,E1 -8370,E2 -8370} C_VEL
LIN {X 0,Y 452.434,Z 785.004,A -85,B 0,C 180,E1 -8371.78,E2 -8371.78} C_VEL
LIN {X 0,Y 452.504,Z 784.192,A -85,B 0,C 180,E1 -8372.671,E2 -8372.671} C_VEL
LIN {X 0,Y 452.472,Z 781.512,A -85,B 0,C 180,E1 -8374.454,E2 -8374.454} C_VEL
LIN {X 0,Y 452.554,Z 778.561,A -85,B 0,C 180,E1 -8375.793,E2 -8375.793} C_VEL
LIN {X 0,Y 452.658,Z 774.738,A -85,B 0,C 180,E1 -8377.135,E2 -8377.135} C_VEL
LIN {X 0,Y 452.839,Z 769.978,A -85,B 0,C 180,E1 -8378.478,E2 -8378.478} C_VEL
LIN {X 0,Y 453.17,Z 763.035,A -85,B 0,C 180,E1 -8380.048,E2 -8380.048} C_VEL
LIN {X 0,Y 453.604,Z 755.823,A -85,B 0,C 180,E1 -8381.393,E2 -8381.393} C_VEL
LIN {X 0,Y 454.011,Z 748.745,A -85,B 0,C 180,E1 -8382.516,E2 -8382.516} C_VEL
LIN {X 0,Y 454.492,Z 740.46,A -85,B 0,C 180,E1 -8383.639,E2 -8383.639} C_VEL
LIN {X 0,Y 455.103,Z 731.736,A -85,B 0,C 180,E1 -8384.647,E2 -8384.647} C_VEL
LIN {X 0,Y 455.681,Z 722.673,A -85,B 0,C 180,E1 -8385.543,E2 -8385.543} C_VEL
LIN {X 0,Y 456.343,Z 713.395,A -85,B 0,C 180,E1 -8386.323,E2 -8386.323} C_VEL
LIN {X 0,Y 456.918,Z 704.05,A -85,B 0,C 180,E1 -8386.992,E2 -8386.992} C_VEL
LIN {X 0,Y 457.498,Z 693.259,A -85,B 0,C 180,E1 -8387.632,E2 -8387.632} C_VEL
LIN {X 0,Y 457.976,Z 682.129,A -85,B 0,C 180,E1 -8388.162,E2 -8388.162} C_VEL
LIN {X 0,Y 458.418,Z 671.6,A -85,B 0,C 180,E1 -8388.549,E2 -8388.549} C_VEL
LIN {X 0,Y 458.758,Z 660.183,A -85,B 0,C 180,E1 -8388.853,E2 -8388.853} C_VEL
LIN {X 0,Y 459.239,Z 630.073,A -85,B 0,C 180,E1 -8389.354,E2 -8389.354} C_VEL
LIN {X 0,Y 459.997,Z 547.984,A -85,B 0,C 180,E1 -8390.656,E2 -8390.656} C_VEL
LIN {X 0,Y 455.164,Z 523.729,A -85,B 0,C 180,E1 -8391.302,E2 -8391.302} C_VEL
LIN {X 0,Y 455.156,Z 522.349,A -85,B 0,C 180,E1 -8391.513,E2 -8391.513} C_VEL
LIN {X 0,Y 456.088,Z 507.583,A -85,B 0,C 180,E1 -8394.585,E2 -8394.585} C_VEL
LIN {X 0,Y 456.46,Z 498.166,A -85,B 0,C 180,E1 -8396.519,E2 -8396.519} C_VEL
LIN {X 0,Y 454.682,Z 488.742,A -85,B 0,C 180,E1 -8398.63,E2 -8398.63} C_VEL
LIN {X 0,Y 453.533,Z 483.234,A -85,B 0,C 180,E1 -8399.957,E2 -8399.957} C_VEL
LIN {X 0,Y 453.489,Z 483.123,A -85,B 0,C 180,E1 -8403.188,E2 -8403.188} C_VEL
LIN {X 0,Y 453.451,Z 483.084,A -85,B 0,C 180,E1 -8406.298,E2 -8406.298} C_VEL
